# B&R Automation Studio project Tmp_Recipe_V1
Automation Studio 4.9.5.36 SP; technology packages: mapp 5.15.0, mappView 5.15.1

## Configuration X20CPU

CPU X20CP1583, AutomationRuntime C4.90, Build 4.1.2, Safety 0.0, Vc V4.52.0

### Task classes (Cpu.sw)
```
Cyclic#8:
  Recipe_01 <- mappRecipe.Recipe_01.prg
  YourTask <- mappRecipe.YourTask.prg
Binaries: udbdef, mvLoader, TCData, arsvcreg, Config, sysconf, ashwd, ashwac, asfw, iomap, Role, User, arconfig, OpcUaMap
Libraries: FileIO, runtime, AsBrStr, standard, AsBrWStr, MpRecipe, MpBase, sys_lib, IecCheck, AsIODiag, AsHttp, AsMem, MpCom, astime, asieccon
```

### Hardware
```
X20CP1583 : X20CP1583 v1.5.0.0
  Connector IF2:
    ActivateDevice = 1
  ConfigurationID = Tmp_Recipe
  UserPartitionSize = 200
  Simulation = 1
  VolatileGlobalPvSize = 300000
  Cyclic8Stack = 20000
  FileDevice1
  FileDeviceName1 = RECIPE_DEVICE
  FileDevicePath1 = F:/
  FileDevice2
  FileDeviceName2 = SIM_DEVICE
  FileDevicePath2 = C:/Temp
  FtpUser1
  FtpUsername1 = br
  FtpUserPassword1 = B9fKGuUbjkGCgEptWUpgQ1eJbLeEvMYqPBCteWUIcCw=
  FtpUserSalt1 = wEo/3/qm
  FTPAccessRight1 = 0
  ActivateSdm = 0
  ActivateOpcUa = 1
  OpcUaInformationModels_PV_Version = 1
```

### Config_0.mprecipecsv - X20CP1583/mappServices/Config_0.mprecipecsv
```
Element gRecipeCsv_01 (Type=mprecipecsv)
```

### Config_1.mprecipexml - X20CP1583/mappServices/Config_1.mprecipexml
```
Element gRecipeXml_01 (Type=mprecipexml)
```

## Logical view

Binary libraries used (declarations not repeated): AsHttp, AsMem, operator, runtime, astime, AsIecCon, FileIO, AsBrStr, AsBrWStr, standard, MpRecipe 5.07.1, MpBase 5.07.0, sys_lib, AsIODiag, MpCom 5.07.1

### Package Logical/Libraries - Global libraries

### Library Logical/Libraries/IecCheck (IEC)
Depends on: sys_lib, AsBrStr

#### IecCheck.fun - Exported functions and function blocks
```iecst
FUNCTION CheckDivSint : SINT (* Check divisor for SINT division *)
	VAR_INPUT
		divisor : SINT;
	END_VAR
END_FUNCTION

FUNCTION CheckDivUsint : USINT (* Check divisor for USINT division *)
	VAR_INPUT
		divisor : USINT;
	END_VAR
END_FUNCTION

FUNCTION CheckDivInt : INT (* Check divisor for INT division *)
	VAR_INPUT
		divisor : INT;
	END_VAR
END_FUNCTION

FUNCTION CheckDivUint : UINT (* Check divisor for UINT division *)
	VAR_INPUT
		divisor : UINT;
	END_VAR
END_FUNCTION

FUNCTION CheckDivDint : DINT (* Check divisor for DINT division *)
	VAR_INPUT
		divisor : DINT;
	END_VAR
END_FUNCTION

FUNCTION CheckDivUdint : UDINT (* Check divisor for UDINT division *)
	VAR_INPUT
		divisor : UDINT;
	END_VAR
END_FUNCTION

FUNCTION CheckDivReal : REAL (* Check divisor for REAL division *)
	VAR_INPUT
		divisor : REAL;
	END_VAR
END_FUNCTION

FUNCTION CheckDivLReal : LREAL (* Check divisor for LREAL division, not available for SG3 and SGC *)
	VAR_INPUT
		divisor : LREAL;
	END_VAR
END_FUNCTION

FUNCTION CheckBounds : DINT (* Check range for array access *)
	VAR_INPUT
		index : DINT;
		lower : DINT;
		upper : DINT;
	END_VAR
END_FUNCTION

FUNCTION CheckRange : DINT (* Check range for enumeration *)
	VAR_INPUT
		value : DINT;
		lower : DINT;
		upper : DINT;
	END_VAR
END_FUNCTION

FUNCTION CheckSignedSubrange : DINT (* Check range for subrange of signed data types *)
	VAR_INPUT
		value : DINT;
		lower : DINT;
		upper : DINT;
	END_VAR
END_FUNCTION

FUNCTION CheckUnsignedSubrange : UDINT (* Check range for subrange of unsigned data types *)
	VAR_INPUT
		value : UDINT;
		lower : UDINT;
		upper : UDINT;
	END_VAR
END_FUNCTION

FUNCTION CheckReadAccess : UDINT (* Check address when reading dynamic variables *)
	VAR_INPUT
		address : UDINT;
	END_VAR
END_FUNCTION

FUNCTION CheckWriteAccess : UDINT (* Check address when writing dynamic variables *)
	VAR_INPUT
		address : UDINT;
	END_VAR
END_FUNCTION

FUNCTION MakeEntry : UDINT (* Makes an entry (log book entry) in the error log book *)
	VAR
		taskname : STRING[30];
		group : USINT;
		status_name : UINT;
		out_text : STRING[80];
	END_VAR
	VAR_INPUT
		number : UINT;
		index : DINT;
		text : STRING[50];
	END_VAR
END_FUNCTION
```

#### IecCheck.st - Implementation file
```iecst
(* Check divisor for SINT division *)
FUNCTION CheckDivSint
	IF divisor=0 THEN
		CheckDivSint:=1;
		MakeEntry(55555,divisor,'CheckDivSint');
	ELSE
		CheckDivSint:=divisor;
	END_IF
END_FUNCTION

(* Check divisor for USINT division *)
FUNCTION CheckDivUsint
	IF divisor=0 THEN
		CheckDivUsint:=1;
		MakeEntry(55555,divisor,'CheckDivUsint');
	ELSE
		CheckDivUsint:=divisor;
	END_IF
END_FUNCTION

(* Check divisor for INT division *)
FUNCTION CheckDivInt
	IF divisor=0 THEN
		CheckDivInt:=1;
		MakeEntry(55555,divisor,'CheckDivInt');
	ELSE
		CheckDivInt:=divisor;
	END_IF
END_FUNCTION

(* Check divisor for UINT division *)
FUNCTION CheckDivUint
	IF divisor=0 THEN
		CheckDivUint:=1;
		MakeEntry(55555,divisor,'CheckDivUint');
	ELSE
		CheckDivUint:=divisor;
	END_IF
END_FUNCTION

(* Check divisor for DINT division *)
FUNCTION CheckDivDint
	IF divisor=0 THEN
		CheckDivDint:=1;
		MakeEntry(55555,divisor,'CheckDivDint');
	ELSE
		CheckDivDint:=divisor;
	END_IF
END_FUNCTION

(* Check divisor for UDINT division *)
FUNCTION CheckDivUdint
	IF divisor=0 THEN
		CheckDivUdint:=1;
		MakeEntry(55555,divisor,'CheckDivUdint');
	ELSE
		CheckDivUdint:=divisor;
	END_IF
END_FUNCTION

(* Check divisor for REAL division *)
FUNCTION CheckDivReal
	IF divisor=0 THEN
		CheckDivReal:=1;
		MakeEntry(55555,0,'CheckDivReal');
	ELSE
		CheckDivReal:=divisor;
	END_IF
END_FUNCTION

(* Check divisor for LREAL division *)
FUNCTION CheckDivLReal
	IF divisor=0 THEN
		CheckDivLReal:=1;
		MakeEntry(55555,0,'CheckDivLReal');
	ELSE
		CheckDivLReal:=divisor;
	END_IF
END_FUNCTION

(* Check range for array access *)
FUNCTION CheckBounds
	IF index < lower THEN
		CheckBounds := lower;
		MakeEntry(55555,index,'CheckBounds');
	ELSIF index > upper THEN
		CheckBounds := upper;
		MakeEntry(55555,index,'CheckBounds');
	ELSE
		CheckBounds := index;
	END_IF
END_FUNCTION

(* Check range for enumeration *)
FUNCTION CheckRange
	IF value < lower THEN
		CheckRange := lower;
		MakeEntry(55555,value,'CheckRange');
	ELSIF value > upper THEN
		CheckRange := upper;
		MakeEntry(55555,value,'CheckRange');
	ELSE
		CheckRange := value;
	END_IF
END_FUNCTION

(* Check range for subrange of signed data types *)
FUNCTION CheckSignedSubrange
	IF value < lower THEN
		CheckSignedSubrange := lower;
		MakeEntry(55555,value,'CheckSignedSubrange');
	ELSIF value > upper THEN
		CheckSignedSubrange := upper;
		MakeEntry(55555,value,'CheckSignedSubrange');
	ELSE
		CheckSignedSubrange := value;
	END_IF
END_FUNCTION

(* Check range for subrange of unsigned data types *)
FUNCTION CheckUnsignedSubrange
	IF value < lower THEN
		CheckUnsignedSubrange := lower;
		MakeEntry(55555,value,'CheckUnsignedSubrange');
	ELSIF value > upper THEN
		CheckUnsignedSubrange := upper;
		MakeEntry(55555,value,'CheckUnsignedSubrange');
	ELSE
		CheckUnsignedSubrange := value;
	END_IF
END_FUNCTION

(* Check address when reading dynamic variables *)
FUNCTION CheckReadAccess
	IF address=0 THEN
		(* TODO: Insert an appropriate code, see AutomationStudio help for further information *)
		MakeEntry(55555,address,'Read from NULL');
	END_IF

	CheckReadAccess:=0;
END_FUNCTION

(* Check address when writing dynamic variables *)
FUNCTION CheckWriteAccess
	IF address=0 THEN
		(* TODO: Insert an appropriate code, see AutomationStudio help for further information *)
		MakeEntry(55555,address,'Write to NULL');
	END_IF

	CheckWriteAccess:=0;
END_FUNCTION

(* Makes an entry (log book entry) in the error log book *)
FUNCTION MakeEntry
		status_name := ST_name(0,ADR(taskname),ADR(group));

		brsstrcpy(ADR(out_text),ADR(text));
		brsstrcat(ADR(out_text),ADR(' > in task > '));
  		brsstrcat(ADR(out_text),ADR(taskname));
		MakeEntry := ADR(out_text);
		ERRxfatal(number,index,ADR(out_text));
END_FUNCTION
```

- Visualisation Logical/mappView (not shown)

### RecTypes.typ
```iecst
(*------------------------------------------------------------------------------------------------------------------------------------------------------------------------------------------------------------------------*)
(*Global enumerations*)

TYPE
	recSTATE :
		( (*Recipe management state machine*)
		REC_WAIT,
		REC_REG_NAME,
		REC_REG_VAR,
		REC_CREATE_DIR,
		REC_READ_DIR,
		REC_READ_DIR_1,
		REC_READ_DIR_2,
		REC_READ_DIR_3,
		REC_GEN_FILE_NAME,
		REC_LOAD_SAVE,
		REC_DELETE,
		REC_RENAME,
		REC_VIEW,
		REC_DOWNLOAD,
		REC_DOWNLOAD_1,
		REC_DOWNLOAD_2,
		REC_DOWNLOAD_3,
		REC_DOWNLOAD_4,
		REC_UPLOAD,
		REC_UPLOAD_1,
		REC_UPLOAD_2,
		REC_UPLOAD_3,
		REC_UPLOAD_4,
		REC_UPLOAD_5,
		REC_UPLOAD_6,
		REC_ERROR
		);
	recTYPE :
		(
		typeCSV,
		typeXML
		);
END_TYPE

(*------------------------------------------------------------------------------------------------------------------------------------------------------------------------------------------------------------------------*)
(*Global structure*)

TYPE
	recERR : 	STRUCT  (*Recipe management error structure*)
		Text : WSTRING[200]; (* Error text *)
		No : DINT; (* Error number *)
		State : recSTATE; (* Error step *)
	END_STRUCT;
	recCMD : 	STRUCT  (*Recipe management command structure*)
		Init : BOOL := TRUE; (*Init recipes managment*)
		New : BOOL; (*Create new recipe*)
		Load : BOOL; (*Load recipe*)
		Save : BOOL; (*Save recipe*)
		View : BOOL; (*View recipe*)
		Rename : BOOL; (*Rename recipe*)
		Delete : BOOL; (*Delete recipe*)
		Download : BOOL; (*Download recipe*)
		Upload : BOOL; (*Upload recipe*)
		ErrorReset : BOOL; (*Reset pending errors*)
	END_STRUCT;
	recPAR : 	STRUCT  (*Recipe management parameter structure*)
		RecipeName : WSTRING[REC_NAME_LENGTH]; (*Recipe name*)
		RecipeNameNew : WSTRING[REC_NAME_LENGTH]; (*New recipe name*)
		RecipeID : STRING[REC_NAME_LENGTH]; (*File name of the recipe*)
		Initialized : BOOL; (*Indicates that recipe management was initialized*)
		VisuSlotID : USINT; (*ID for connected web connection*)
		VisuEnableCommand : BOOL;
	END_STRUCT;
	recDAT : 	STRUCT  (*Recipe management data structure*)
		RecipeNames : ARRAY[0..REC_REC_NUM]OF WSTRING[REC_NAME_LENGTH]; (*Recipe unicode names*)
		RecipeIDs : ARRAY[0..REC_REC_NUM]OF STRING[REC_NAME_LENGTH]; (*File name of the recipes*)
		RecipeNum : UINT; (*Number of recipes*)
		Status : WSTRING[100]; (*Shows the result of the last command*)
	END_STRUCT;
	recVIS : 	STRUCT  (*Recipe management visualization structure*)
		RecipeNames : ARRAY[0..REC_REC_NUM]OF WSTRING[REC_VIS_LENGTH]; (*Recipe names as mappView data provider*)
		RecipeNum : UINT; (*Number of visible recipes*)
		RecipeFilter : WSTRING[REC_NAME_LENGTH]; (*Only show recipes that fit this pattern*)
		RecipeSelect : WSTRING[REC_NAME_LENGTH]; (*Select recipe in listbox after command new or rename*)
		DownloadFileUrl : STRING[REC_NAME_LENGTH]; (*URL used with recipe download*)
		UploadOverwriteRequest : BOOL; (*Show message box to overwrite file*)
		UploadOverwriteResponse : USINT; (*Response from message box overwrite file*)
		ReloadUpload : BOOL; (*Reload upload button*)
		RecipeDoubleClick : USINT; (*Track double click event*)
		ViewFilePath : STRING[REC_VIS_LENGTH]; (*Full path for viewing file*)
		ViewFile : BOOL; (*Trigger that opens the fly out window when viewing recipes*)
		ShowMessageBoxError : BOOL; (*Show message box on error*)
	END_STRUCT;
	recMAIN : 	STRUCT  (*Recipe management main structure*)
		CMD : recCMD; (* Command structure *)
		PAR : recPAR; (* Parameter structure *)
		DAT : recDAT; (*Data structure*)
		VIS : ARRAY[0..REC_MAX_CLIENTS_ID]OF recVIS; (*Visualization structure*)
		ERR : recERR; (* Error structure *)
	END_STRUCT;
END_TYPE
```

### RecVariables.var
```iecst
(*------------------------------------------------------------------------------------------------------------------------------------------------------------------------------------------------------------------------*)
(*Configuration for recipe managment*)
VAR CONSTANT
	REC_USE_UNICODE : BOOL := FALSE; (*Use standard strings for recipe name when false, use unicode strings for recipe name when true*)
	REC_SORT_NUMERIC : BOOL := FALSE; (*Sort recipe names as numeric values instead of alphabetic*)
	REC_RECIPE_TYPE : recTYPE := typeCSV; (*Type of recipe (CSV / XML)*)
END_VAR
VAR
	REC_MPLINK : {REDUND_UNREPLICABLE} STRING[80] := 'gRecipeCsv_01'; (*mappRecipe link name from configuration view. User gRecipeCsv_01 for CSV and gRecipeXml_01 for XML in this demo*)
END_VAR
VAR CONSTANT
	REC_DEVICE : STRING[80] := 'RECIPE_DEVICE'; (*Device name for the recipe data defined under File Devices in the CPU configuration*)
	REC_DIRECTORY : STRING[80] := 'Recipe_01'; (*Directory where the recipes are stored*)
	REC_THIS_TASK : STRING[40] := 'Recipe_01'; (*Name of this task and the global variables structure*)
	REC_REC_NUM : USINT := 100; (*Maximum number of recipes*)
	REC_VAR_NUM : USINT := 10; (*Maximum number of variables that can be registered*)
	REC_NAME_LENGTH : USINT := 40; (*Maximum length for a recipe name*)
	REC_UPLOAD_DOWNLOAD_SIZE : UDINT := 100000; (*Maximum size of memory allocated for uploading and downloading files*)
	REC_VIS_LENGTH : USINT := 120; (*Make this REC_NAME_LENGTH  x3*)
	REC_MAX_CLIENTS_ID : USINT := 2; (*Highest client ID for concurrent web client connections. Do not change this number.*)
END_VAR
VAR
	REC_VIEW_FILTER : ARRAY[0..9] OF STRING[5] := ['csv','xml',8('')]; (*Files extensions than can be used with the view command*)
END_VAR
(*------------------------------------------------------------------------------------------------------------------------------------------------------------------------------------------------------------------------*)
(*Add you variables to this list*)
VAR
	REC_VAR_LIST : ARRAY[1..REC_VAR_NUM] OF STRING[100] := ['YourTask:MaschineData','YourTask:ProductID','YourTask:CustomerID',7('')]; (*List of variables to be inlcuded in a recipe*)
	Recipe_01 : recMAIN; (*Global recipe structure. The name must match the task name of the recipe managment.*)
END_VAR
```

### Program Logical/mappRecipe/Recipe_01 (IEC)

#### Init.st - Init and local configuration
```iecst
// --------------------------------------------------------------------------------------------------------------------
//	Function:	Recipe management with mappRecipe
//  Version:	0.7
//	Changed:	08.05.2020
// --------------------------------------------------------------------------------------------------------------------

PROGRAM _INIT
	// ----------------------------------------------------------------------------------------
	// The following settings can be adjusted
	IF(DiagCpuIsSimulated()) THEN
		DeviceName 	:= 'SIM_DEVICE';						// Device name from the CPU configuration for simulation
	ELSE
		DeviceName 	:= REC_DEVICE;							// Device name from the CPU configuration for X20CPU
	END_IF

	// ----------------------------------------------------------------------------------------
	// Dont change anything below this line
	// ----------------------------------------------------------------------------------------

	// ----------------------------------------------------------------------------------------
	// Get mapp link information
	MpComGetLink_0.Enable := TRUE;
	MpComGetLink_0.ComponentName := ADR(REC_MPLINK);
	MpComGetLink_0();
	IF(MpComGetLink_0.Error) THEN
	END_IF

	// ----------------------------------------------------------------------------------------
	// Make sure global variable structure and task name are correct
	taskStatus := ST_ident(ADR(REC_THIS_TASK), taskGroup, ADR(taskID));
	pvStatus := PV_xgetadr(ADR(REC_THIS_TASK), ADR(pvADR), ADR(pvLEN));
	// Connect global and local structure
	IF(pvStatus = 0) THEN
		RECIPE ACCESS pvADR;
		brsmemset(ADR(RECIPE.ERR), 0 , SIZEOF(RECIPE.ERR));
		RECIPE.PAR.Initialized := FALSE;
	END_IF

	// ----------------------------------------------------------------------------------------
	// Allocate memory for file upload and download
	AsMemPartCreate_0.enable	:= TRUE;
	AsMemPartCreate_0.len		:= REC_UPLOAD_DOWNLOAD_SIZE;
	AsMemPartCreate_0();
	IF AsMemPartCreate_0.status <> 0 THEN
		rec_state := CreateError(ADR(RECIPE), ERR_MEM_ALLOC, "file upload and download memory alloc failed", rec_state);
	ELSE
		AsMemPartAllocClear_0.enable	:= TRUE;
		AsMemPartAllocClear_0.ident		:= AsMemPartCreate_0.ident;
		AsMemPartAllocClear_0.len		:= REC_UPLOAD_DOWNLOAD_SIZE;
		AsMemPartAllocClear_0();
		IF AsMemPartCreate_0.status <> 0 THEN
			rec_state := CreateError(ADR(RECIPE), ERR_MEM_ALLOC, "file upload and download memory clear failed", rec_state);
		END_IF
	END_IF

	// ----------------------------------------------------------------------------------------
	// Generate HTML messages for web upload
	upload_response	:= '<html><body><form action="/uploadA.html" name="form_upload" method="post" enctype="multipart/form-data" >
	<label for="file-upload" style="font-weight:bold;font-family: sans-serif;font-size:16px;padding:15px 50px;10px;10px;" class="custom-file-upload">Upload</label>
	<input type="file" id="file-upload" style="display:none;" onchange="form.submit()" name="file_selected" content-type="application/octet-stream" />
	</form><body></html> ';
	WebServiceUpload.pServiceName := ADR('uploadA.html');
END_PROGRAM
```

#### Main.st - Cyclic code
```iecst
// --------------------------------------------------------------------------------------------------------------------********
//	Cylic task for recipe management
//	Version 0.7
//	Changed 08.05.2020
// --------------------------------------------------------------------------------------------------------------------********

// --------------------------------------------------------------------------------------------------------------------********
// Cyclic task
// --------------------------------------------------------------------------------------------------------------------********
PROGRAM _CYCLIC
	// --------------------------------------------------------------------------------------------------------------------
	// Make sure task name and global structure correct
	IF(pvStatus <> 0) THEN
		RETURN;
	END_IF
	IF(taskStatus <> 0) THEN
		rec_state := CreateError(ADR(RECIPE), ERR_REC_TASK_NAME, "Task name is incorrect", rec_state);
		RETURN;
	END_IF

	// --------------------------------------------------------------------------------------------------------------------
	// Make sure we dont exceed maximum number of web clients
	IF(RECIPE.PAR.VisuSlotID > REC_MAX_CLIENTS_ID) THEN
		rec_state := CreateError(ADR(RECIPE), ERR_REC_TOO_MANY_CLIENTS, "More than 3 clients try to connect to recipe managment", rec_state);
		RETURN;
	END_IF

	// --------------------------------------------------------------------------------------------------------------------
	// Cyclic function calls
	MpRecipeCsv_0();
	MpRecipeXml_0();

	// ----------------------------------------------------------------------------------------
	// Web service driver for file upload
	WebServiceUpload.enable 			:= TRUE;
	WebServiceUpload.option 			:= httpOPTION_HTTP_11 + httpOPTION_SERVICE_TYPE_NAME;
	WebServiceUpload.pRequestData  		:= AsMemPartAllocClear_0.mem;
	WebServiceUpload.requestDataSize 	:= REC_UPLOAD_DOWNLOAD_SIZE;
	WebServiceUpload.pResponseData 		:= ADR(upload_response);
	WebServiceUpload.responseDataLen 	:= brsstrlen(ADR(upload_response));
	WebServiceUpload();

	// Reset send command
	IF(WebServiceUpload.send = TRUE)  THEN
		WebServiceUpload.send := FALSE;
	// Send response when page is loaded or data is posted
	ELSIF(WebServiceUpload.status = ERR_OK AND WebServiceUpload.send = FALSE) THEN
		WebServiceUpload.send := TRUE;
	// New upload data arrived
	ELSIF(WebServiceUpload.send = FALSE AND WebServiceUpload.requestDataLen > 0 AND RECIPE.CMD.Upload = FALSE) THEN
		// Add delay so that upload can finish
		upload_delay.PT := WebServiceUpload.requestDataLen/100000*5;
		upload_delay.IN := TRUE;
		upload_delay();
	END_IF
	// Check new uploaded data
	IF(upload_delay.Q AND RECIPE.CMD.Upload = FALSE) THEN
		upload_delay.IN := FALSE;
		upload_delay();
		RECIPE.CMD.Upload := TRUE;
	END_IF

	// --------------------------------------------------------------------------------------------------------------------****
	// Recipe management state machine
	// --------------------------------------------------------------------------------------------------------------------****
	CASE rec_state OF
		// --------------------------------------------------------------------------------------------------------------------
		// Wait for command
		// --------------------------------------------------------------------------------------------------------------------
		REC_WAIT:
			// --------------------------------------------------------------------------------------------------------------------
			// Track filter change and data refresh
			IF ((brwcscmp(ADR(RecipeFilterOld[VisuSlotID]), ADR(RECIPE.VIS[VisuSlotID].RecipeFilter)) <> 0) OR (RecipeNumOld[VisuSlotID] <> RECIPE.DAT.RecipeNum)) THEN
				brsmemset(ADR(RECIPE.VIS[VisuSlotID].RecipeNames), 0, SIZEOF(RECIPE.VIS[VisuSlotID].RecipeNames));
				idy := 0;
				IF(RECIPE.DAT.RecipeNum > 0) THEN
					FOR idx:=0 TO RECIPE.DAT.RecipeNum - 1 DO
						// --------------------------------------------------------------------------------
						// Verify that file name contains filter
						IF (brwcslen(ADR(RECIPE.VIS[VisuSlotID].RecipeFilter)) = 0 OR IsInstrW(ADR(RECIPE.DAT.RecipeNames[idx]), ADR(RECIPE.VIS[VisuSlotID].RecipeFilter))) THEN
							WString2DataProvider(ADR(RECIPE.DAT.RecipeNames[idx]), ADR(tmpWStr1));
							RECIPE.VIS[VisuSlotID].RecipeNames[idy] := tmpWStr1;
							idy := idy + 1;
						END_IF
					END_FOR;
					brwcscpy(ADR(RecipeFilterOld[VisuSlotID]), ADR(RECIPE.VIS[VisuSlotID].RecipeFilter));
				END_IF
				RecipeNumOld[VisuSlotID] := RECIPE.DAT.RecipeNum;
				RECIPE.VIS[VisuSlotID].RecipeNum := idy;
			END_IF

			// ------------------------------------------------------------------------------------------------
			// Handle double click for file open
			IF(RECIPE.VIS[VisuSlotID].RecipeDoubleClick > 0) THEN
				DoubleClickRecipeName[VisuSlotID].PT := 50;
				DoubleClickRecipeName[VisuSlotID].IN := TRUE;
				DoubleClickRecipeName[VisuSlotID]();
				// Open selected file
				IF(RECIPE.VIS[VisuSlotID].RecipeDoubleClick > 1) THEN
					DoubleClickRecipeName[VisuSlotID].IN := FALSE;
					DoubleClickRecipeName[VisuSlotID]();
					RECIPE.VIS[VisuSlotID].RecipeDoubleClick := 0;
					RECIPE.PAR.VisuSlotID := VisuSlotID;
					RECIPE.PAR.RecipeName := RECIPE.VIS[VisuSlotID].RecipeSelect;
					RECIPE.CMD.View := TRUE;
				END_IF
			END_IF
			IF(DoubleClickRecipeName[VisuSlotID].Q) THEN
				DoubleClickRecipeName[VisuSlotID].IN := FALSE;
				DoubleClickRecipeName[VisuSlotID]();
				IF(RECIPE.VIS[VisuSlotID].RecipeDoubleClick > 0) THEN
					RECIPE.VIS[VisuSlotID].RecipeDoubleClick := RECIPE.VIS[VisuSlotID].RecipeDoubleClick - 1;
				END_IF
			END_IF

			// Cylce through the client web seesions
			VisuSlotID := VisuSlotID + 1;
			IF(VisuSlotID > REC_MAX_CLIENTS_ID) THEN
				VisuSlotID := 0;
			END_IF

			// --------------------------------------------------------------------------------------------------------------------
			// Disable buttons in visualization when number of recipes is 0
			IF(RECIPE.DAT.RecipeNum = 0) THEN
				RECIPE.PAR.VisuEnableCommand := FALSE;
			ELSE
				RECIPE.PAR.VisuEnableCommand := TRUE;
			END_IF

			// ----------------------------------------------------------------------------------------
			// Reset error reset
			MpRecipeCsv_0.ErrorReset := FALSE;
			MpRecipeXml_0.ErrorReset := FALSE;
			MpRecipeRegPar_0.ErrorReset := FALSE;

			// ----------------------------------------------------------------------------------------
			// Command init/refresh
			IF (RECIPE.CMD.Init = TRUE) THEN
				// Reset data structure and trigger name refresh for vis
				brsmemset(ADR(RECIPE.DAT), 0, SIZEOF(RECIPE.DAT));
				brsmemset(ADR(RecipeIDs), 0, SIZEOF(RecipeIDs));
				brsmemset(ADR(RecipeNumOld), 16#FF, SIZEOF(RecipeNumOld));
				// Skip variable binding if already initialized
				IF(MpRecipeRegPar_1[1].PVName <> 0) THEN
					rec_state := REC_READ_DIR;
				ELSE
					// Register recipe name variable first if unicode is used
					IF(REC_USE_UNICODE) THEN
						rec_state := REC_REG_NAME;
					ELSE
						rec_state := REC_REG_VAR;
					END_IF
					pvCnt := 1;
				END_IF
			// ----------------------------------------------------------------------------------------
			// Command new recipe
			ELSIF (RECIPE.CMD.New = TRUE AND RECIPE.PAR.RecipeName <> "") THEN
				// Show current state
				animation := WorkingStatus(ADR(RECIPE), ADR("creating recipe..."), animation);
				// Verify that we still have space in list
				IF (RECIPE.DAT.RecipeNum > REC_REC_NUM) THEN
					rec_state := CreateError(ADR(RECIPE), ERR_REC_REC_NUM, "maximum number of recipes reached", rec_state);
					RETURN;
				END_IF
				// Make sure recipe does not already exist
				IF(FindRecName(ADR(RECIPE), RECIPE.PAR.RecipeName) <> REC_DOES_NOT_EXIST) THEN
					tmpWStr1 := "recipe name ";
					brwcscat(ADR(tmpWStr1), ADR(RECIPE.PAR.RecipeName));
					brwcscat(ADR(tmpWStr1), ADR(" already exists"));
					rec_state := CreateError(ADR(RECIPE), ERR_REC_NAME_EXISTS, tmpWStr1, rec_state);
					RETURN;
				END_IF
				// Reset selected recipe, copy recipe name to local variable
				RECIPE.VIS[RECIPE.PAR.VisuSlotID].RecipeSelect := "";
				rec_state := REC_GEN_FILE_NAME;
			// ----------------------------------------------------------------------------------------
			// Command load recipe
			ELSIF (RECIPE.CMD.Load = TRUE AND RECIPE.PAR.RecipeName <> "") THEN
				// Show current state
				animation := WorkingStatus(ADR(RECIPE), ADR("loading recipe..."), animation);
				// Copy recipe name to local variable
				rec_state := REC_GEN_FILE_NAME;
				// ----------------------------------------------------------------------------------------
			// Command save recipe
			ELSIF (RECIPE.CMD.Save = TRUE AND (RECIPE.PAR.RecipeName <> "" OR RECIPE.PAR.RecipeNameNew <> "")) THEN
				// Show current state
				animation := WorkingStatus(ADR(RECIPE), ADR("saving recipe..."), animation);
				IF(RECIPE.PAR.RecipeName = "") THEN
					RECIPE.PAR.RecipeName := RECIPE.PAR.RecipeNameNew;
				END_IF
				// Copy recipe name to local variable
				rec_state := REC_GEN_FILE_NAME;
			// ----------------------------------------------------------------------------------------
			// Command view recipe
			ELSIF (RECIPE.CMD.View = TRUE AND RECIPE.PAR.RecipeName <> "") THEN
				// Copy recipe name to local variable
				rec_state := REC_GEN_FILE_NAME;
			// ----------------------------------------------------------------------------------------
			// Command delete recipe
			ELSIF (RECIPE.CMD.Delete = TRUE AND RECIPE.PAR.RecipeName <> "") THEN
				// Show current state, copy recipe name to local variable
				animation := WorkingStatus(ADR(RECIPE), ADR("deleting recipe..."), animation);
				rec_state := REC_GEN_FILE_NAME;
			// ----------------------------------------------------------------------------------------
			// Command download recipe
			ELSIF (RECIPE.CMD.Download = TRUE AND RECIPE.PAR.RecipeName <> "") THEN
				// Show current state, copy recipe name to local variable
				animation := WorkingStatus(ADR(RECIPE), ADR("downloading recipe..."), animation);
				RECIPE.VIS[RECIPE.PAR.VisuSlotID].DownloadFileUrl := '';
				rec_state := REC_GEN_FILE_NAME;
			// ----------------------------------------------------------------------------------------
			// Command upload recipe
			ELSIF (RECIPE.CMD.Upload = TRUE) THEN
				// Make sure that unicode support is turned off
				IF(REC_USE_UNICODE = FALSE) THEN
					// Show current state, copy recipe name to local variable
					animation := WorkingStatus(ADR(RECIPE), ADR("uploading recipe..."), animation);
					rec_state := REC_UPLOAD;
				ELSE
					rec_state := CreateError(ADR(RECIPE), ERR_UNICODE_UPLOAD, "upload is not supported when using unicode recipes", rec_state);
				END_IF
			// ----------------------------------------------------------------------------------------
			// Rename recipe
			ELSIF (RECIPE.CMD.Rename = TRUE AND RECIPE.PAR.RecipeName <> "" AND RECIPE.PAR.RecipeNameNew <> "") THEN
				// Show current state
				animation := WorkingStatus(ADR(RECIPE), ADR("renaming recipe..."), animation);
				// Make sure new recipe name does not already exist
				IF(FindRecName(ADR(RECIPE), RECIPE.PAR.RecipeNameNew) <> REC_DOES_NOT_EXIST) THEN
					tmpWStr1 := "new recipe name ";
					brwcscat(ADR(tmpWStr1), ADR(RECIPE.PAR.RecipeNameNew));
					brwcscat(ADR(tmpWStr1), ADR(" already exists"));
					rec_state := CreateError(ADR(RECIPE), ERR_REC_NAME_EXISTS, tmpWStr1, rec_state);
					RETURN;
				END_IF
				// Reset selected recipe, copy recipe name to local variable
				brsmemset(ADR(RecipeNumOld), 16#FF, SIZEOF(RecipeNumOld));
				RECIPE.VIS[RECIPE.PAR.VisuSlotID].RecipeSelect := "";
				RecipeNameNew := RECIPE.PAR.RecipeNameNew;
				rec_state := REC_GEN_FILE_NAME;
			END_IF
			RecipeName := RECIPE.PAR.RecipeName;

			// ----------------------------------------------------------------------------------------
			// Check parameters
			IF (RECIPE.CMD.Init OR RECIPE.CMD.New OR RECIPE.CMD.Load OR RECIPE.CMD.Save OR RECIPE.CMD.Rename OR RECIPE.CMD.Delete OR RECIPE.CMD.View) THEN
				// Make sure recipe mangament was intialized
				IF (NOT RECIPE.CMD.Init AND NOT RECIPE.PAR.Initialized) THEN
					rec_state := CreateError(ADR(RECIPE), ERR_REC_NOT_INITIALIZED, "recipe management is not initiialized", rec_state);
				END_IF
				// Make sure recipe name is valid
				IF((RECIPE.CMD.New OR RECIPE.CMD.Load OR RECIPE.CMD.Save OR RECIPE.CMD.Rename OR RECIPE.CMD.Delete OR RECIPE.CMD.View) AND RecipeName = "") THEN
					rec_state := CreateError(ADR(RECIPE), ERR_REC_NAME_EMPTY, "recipe name is empty", rec_state);
				END_IF
				// Make sure new recipe name is valid
				IF((RECIPE.CMD.Rename) AND RecipeNameNew = "") THEN
					rec_state := CreateError(ADR(RECIPE), ERR_REC_NAME_EMPTY, "new recipe name is empty", rec_state);
				END_IF
				// Make sure device name is valid
				IF(DeviceName = '') THEN
					rec_state := CreateError(ADR(RECIPE), ERR_REC_DEV_NAME_EMPTY, "device name is empty", rec_state);
				END_IF
				// Make sure variable name has at least one entry
				IF(REC_VAR_LIST[1] = '') THEN
					rec_state := CreateError(ADR(RECIPE), ERR_REC_VAR_NAME_EMPTY, "variable name is empty", rec_state);
				END_IF

				RECIPE.PAR.VisuEnableCommand := FALSE;
			END_IF
		// --------------------------------------------------------------------------------------------------------------------
		// Register recipe name
		// --------------------------------------------------------------------------------------------------------------------
		REC_REG_NAME:
			// Generate string for local recipe name
			tmpStr1 := REC_THIS_TASK;
			brsstrcat(ADR(tmpStr1), ADR(':RecipeName'));

			MpRecipeRegPar_0.Enable := TRUE;
			MpRecipeRegPar_0.MpLink := ADR(MpComGetLink_0.MpLink);
			MpRecipeRegPar_0.PVName := ADR(tmpStr1);
			MpRecipeRegPar_0.Category := ADR(REC_THIS_TASK);

			// ----------------------------------------------------------------------------------------
			// OK
			IF (NOT MpRecipeRegPar_0.Active AND NOT MpRecipeRegPar_0.Error) THEN
				rec_state := REC_REG_VAR;
			// Error
			ELSIF (MpRecipeRegPar_0.Error) THEN
				rec_state := CreateError(ADR(RECIPE), MpRecipeRegPar_0.StatusID, "error trying to register recipe name", rec_state);
			END_IF
		// --------------------------------------------------------------------------------------------------------------------
		// Register variable structure
		// --------------------------------------------------------------------------------------------------------------------
		REC_REG_VAR:
			MpRecipeRegPar_1[pvCnt].Enable := TRUE;
			MpRecipeRegPar_1[pvCnt].MpLink := ADR(MpComGetLink_0.MpLink);
			MpRecipeRegPar_1[pvCnt].PVName := ADR(REC_VAR_LIST[pvCnt]);
			MpRecipeRegPar_1[pvCnt].Category := ADR(REC_THIS_TASK);

			// ----------------------------------------------------------------------------------------
			// OK
			IF (MpRecipeRegPar_1[pvCnt].Active AND NOT MpRecipeRegPar_1[pvCnt].Error) THEN
				pvCnt := pvCnt + 1;
				// Register next variable
				IF((pvCnt >= SIZEOF(REC_VAR_LIST)/SIZEOF(REC_VAR_LIST[pvCnt])) OR (REC_VAR_LIST[pvCnt] = '')) THEN
					rec_state := REC_CREATE_DIR;
				END_IF
			// Error
			ELSIF (MpRecipeRegPar_1[pvCnt].Error) THEN
				tmpWStr1 := "error trying to register variable name ";
				brwcsconv(ADR(tmpWStr2), ADR(REC_VAR_LIST[pvCnt]), brwU8toUC);
				brwcscat(ADR(tmpWStr1), ADR(tmpWStr2));
				rec_state := CreateError(ADR(RECIPE), MpRecipeRegPar_1[pvCnt].StatusID, tmpWStr1, rec_state);
			END_IF
		// --------------------------------------------------------------------------------------------------------------------
		// Create recipe directory
		// --------------------------------------------------------------------------------------------------------------------
		REC_CREATE_DIR:
			DCreate.enable 	:= TRUE;
			DCreate.pDevice	:= ADR(DeviceName);
			DCreate.pName := ADR(REC_DIRECTORY);
			DCreate();

			// ----------------------------------------------------------------------------------------
			// OK
			IF (DCreate.status = OK OR DCreate.status = fiERR_DIR_ALREADY_EXIST) THEN
				// Reset command and return to wait state
				rec_state := REC_READ_DIR;
			// Error
			ELSIF (DCreate.status <> ERR_FUB_BUSY) THEN
				// File device is wrong
				IF(DCreate.status = fiERR_DEVICE_MANAGER) THEN
					rec_state := CreateError(ADR(RECIPE), DCreate.status, "error creating recipe directory, check file device name", rec_state);
				ELSE
					rec_state := CreateError(ADR(RECIPE), DCreate.status, "error creating recipe directory", rec_state);
				END_IF
			END_IF
		// --------------------------------------------------------------------------------------------------------------------
		// Read directory information
		// --------------------------------------------------------------------------------------------------------------------
		REC_READ_DIR:
			// Show current state
			animation := WorkingStatus(ADR(RECIPE), ADR("reading recipes..."), animation);
			// ----------------------------------------------------------------------------------------
			// Clear all entrys
			brsmemset(ADR(RECIPE.DAT), 0, SIZEOF(RECIPE.DAT));
			RECIPE.DAT.RecipeNum := 0;
			// ----------------------------------------------------------------------------------------
			// Set values and get device dir
			DInfo.enable 	:= TRUE;
			DInfo.pDevice	:= ADR(DeviceName);
			DInfo();

			// ----------------------------------------------------------------------------------------
			// OK
			IF (DInfo.status = OK) THEN
				rec_state := REC_READ_DIR_1;
			ELSIF (DInfo.status = fiERR_DEVICE_MANAGER) THEN
				tmpWStr1 := "file device ";
				brwcsconv(ADR(tmpWStr2), ADR(DeviceName), brwU8toUC);
				brwcscat(ADR(tmpWStr1), ADR(tmpWStr2));
				brwcscat(ADR(tmpWStr1), ADR(" is unavailable"));
				rec_state := CreateError(ADR(RECIPE), DInfo.status, tmpWStr1, rec_state);
			ELSIF (DInfo.status = fiERR_DIR_NOT_EXIST) THEN
				tmpWStr1 := "file ";
				brwcsconv(ADR(tmpWStr2), ADR(REC_DIRECTORY), brwU8toUC);
				brwcscat(ADR(tmpWStr1), ADR(tmpWStr2));
				brwcscat(ADR(tmpWStr1), ADR(" is unavailable"));
				rec_state := CreateError(ADR(RECIPE), DInfo.status, tmpWStr1, rec_state);
				// Error
			ELSIF (DInfo.status <> ERR_FUB_BUSY) THEN
				rec_state := CreateError(ADR(RECIPE), DInfo.status, "error dir info", rec_state);
			END_IF
		// --------------------------------------------------------------------------------------------------------------------
		// Open directory
		// --------------------------------------------------------------------------------------------------------------------
		REC_READ_DIR_1:
			DOpen.enable 	:= TRUE;
			DOpen.pDevice	:= ADR(DeviceName);
			DOpen.pName 	:= ADR(REC_DIRECTORY);
			DOpen();

			// ----------------------------------------------------------------------------------------
			// OK
			IF (DOpen.status = OK) THEN
				rec_state := REC_READ_DIR_2;
			// Create error message for missing directory
			ELSIF (DInfo.status = fiERR_DIR_NOT_EXIST) THEN
				tmpWStr1 := "directory ";
				brwcsconv(ADR(tmpWStr2), ADR(REC_DIRECTORY), brwU8toUC);
				brwcscat(ADR(tmpWStr1), ADR(tmpWStr2));
				brwcscat(ADR(tmpWStr1), ADR(" is unavailable"));
				rec_state := CreateError(ADR(RECIPE), DInfo.status, tmpWStr1, rec_state);
			// Error
			ELSIF (DOpen.status <> ERR_FUB_BUSY) THEN
				rec_state := CreateError(ADR(RECIPE), DOpen.status, "error dir open", rec_state);
			END_IF;
		// --------------------------------------------------------------------------------------------------------------------
		// Read file directory information
		// --------------------------------------------------------------------------------------------------------------------
		REC_READ_DIR_2:
			DRead.enable 	:= TRUE;
			DRead.ident		:= DOpen.ident;
			DRead.pData 	:= ADR(lDirReadData);
			DRead.data_len 	:= SIZEOF(lDirReadData);
			DRead();

			// ----------------------------------------------------------------------------------------
			// OK
			IF (DRead.status = OK AND lDirReadData.Mode = fiFILE) THEN
				animation := WorkingStatus(ADR(RECIPE), ADR("initializing recipe managment..."), animation);
				// Make sure file name does not exceed maximum string size
				IF (brsstrlen(ADR(lDirReadData.Filename)) < REC_NAME_LENGTH) THEN
					// Copy dir info to string
					brsmemset(ADR(RECIPE.PAR.RecipeID), 0, SIZEOF(RECIPE.PAR.RecipeID));
					brsstrcpy(ADR(RECIPE.PAR.RecipeID), ADR(lDirReadData.Filename));
					// Make sure file extension is CSV or XML
					IF(brsstrlen(ADR(RECIPE.PAR.RecipeID)) > 4 AND ((REC_RECIPE_TYPE = typeCSV AND brsmemcmp(ADR(RECIPE.PAR.RecipeID) + (brsstrlen(ADR(RECIPE.PAR.RecipeID)) - 4), ADR('.csv'), 4) = 0) OR (REC_RECIPE_TYPE = typeXML AND brsmemcmp(ADR(RECIPE.PAR.RecipeID) + (brsstrlen(ADR(RECIPE.PAR.RecipeID)) - 4), ADR('.xml'), 4) = 0))) THEN
						brsmemset(ADR(RECIPE.PAR.RecipeID) + (brsstrlen(ADR(RECIPE.PAR.RecipeID)) - 4), 0, 4);
						// ------------------------------------------------------------------------------------
						// Verify that we still have space in list
						IF (RECIPE.DAT.RecipeNum <= REC_REC_NUM) THEN
							// --------------------------------------------------------------------
							// Read recipe name from recipe data in next rec_state when using unicode
							IF(REC_USE_UNICODE) THEN
								RecipeIDs[brsatoi(ADR(RECIPE.PAR.RecipeID))] := TRUE;
								rec_state := REC_GEN_FILE_NAME;
								// Generate recipe name from file name
							ELSE
								brwcsconv(ADR(RecipeName), ADR(RECIPE.PAR.RecipeID), brwU8toUC);
								// Generate ASCII data, insert recipe into list
								InsertRecName(ADR(RECIPE), RecipeName, RECIPE.PAR.RecipeID);
							END_IF
							// Error
						ELSE
							rec_state := CreateError(ADR(RECIPE), ERR_REC_REC_NUM, "maximum number of recipes reached", rec_state);
						END_IF
					END_IF
				ELSE
					has_oversized_items := TRUE;
				END_IF
			// Last entry reached
			ELSIF (DRead.status = fiERR_NO_MORE_ENTRIES) THEN
				rec_state := REC_READ_DIR_3;
			// Error
			ELSIF (DRead.status <> ERR_FUB_BUSY AND DRead.status <> OK) THEN
				rec_state := CreateError(ADR(RECIPE), DRead.status, "error recipe list read", rec_state);
			END_IF
		// --------------------------------------------------------------------------------------------------------------------
		// Close directory information
		// --------------------------------------------------------------------------------------------------------------------
		REC_READ_DIR_3:
			DClose.enable 	:= TRUE;
			DClose.ident	:= DOpen.ident;
			DClose();

			// ----------------------------------------------------------------------------------------
			// OK
			IF (DClose.status = OK) THEN
				// Reset command and return to wait state
				RECIPE.DAT.Status := "initializing complete";
				RECIPE.CMD.Init	:= FALSE;
				RECIPE.PAR.RecipeID := '';
				RECIPE.PAR.Initialized := TRUE;
				DClose.ident	:= 0;
				// Create error message for oversized items
				IF(has_oversized_items) THEN
					rec_state := CreateError(ADR(RECIPE), ERR_REC_NAME_LENGTH, "one or more recipe names exceeds maximum length", rec_state);
				ELSE
					rec_state := REC_WAIT;
				END_IF
			// Error
			ELSIF (DClose.status <> ERR_FUB_BUSY) THEN
				rec_state := CreateError(ADR(RECIPE), DClose.status, "error dir close", rec_state);
			END_IF
		// --------------------------------------------------------------------------------------------------------------------
		// Generate recipe name	full path and file name
		// --------------------------------------------------------------------------------------------------------------------
		REC_GEN_FILE_NAME:
			// Find recipe entry
			RecipeIndex := FindRecName(ADR(RECIPE), RecipeName);

			// Generate file name when using unicode strings
			IF(REC_USE_UNICODE) THEN
				// Ignore during init process
				IF(NOT RECIPE.CMD.Init) THEN
					// Find empty slot for new recipe
					IF(RECIPE.CMD.New) THEN
						RecipeIndex := 0;
						WHILE (RecipeIDs[RecipeIndex] = TRUE AND RecipeIndex <= REC_REC_NUM) DO
							RecipeIndex := RecipeIndex + 1;
						END_WHILE;
						// Make sure we found empty slot
						IF(RecipeIndex <= REC_REC_NUM AND RecipeIDs[RecipeIndex] = FALSE) THEN
							brsitoa(RecipeIndex, ADR(RECIPE.PAR.RecipeID));
						ELSE
							rec_state := CreateError(ADR(RECIPE), ERR_REC_REC_NUM, "no empty slot found", rec_state);
							RETURN;
						END_IF
						// Find recipe name in list	for all other command
					ELSE
						// Recipe name was found
						IF(RecipeIndex <> REC_DOES_NOT_EXIST) THEN
							RECIPE.PAR.RecipeID := RECIPE.DAT.RecipeIDs[RecipeIndex];
							// Recipe name was lost
						ELSE
							tmpWStr1 := "recipe name was not found ";
							brwcscat(ADR(tmpWStr1), ADR(RecipeName));
							rec_state := CreateError(ADR(RECIPE), ERR_REC_NAME_LOST, tmpWStr1, rec_state);
							RETURN;
						END_IF
					END_IF
				END_IF
			// Use recipe name as file name when using standard strings
			ELSE
				brwcsconv(ADR(RECIPE.PAR.RecipeID), ADR(RecipeName), brwUCtoU8);
			END_IF

			// Generate recipe path and extension
			RecipeFullFileName := REC_DIRECTORY;
			brsstrcat(ADR(RecipeFullFileName), ADR('/'));
			brsstrcat(ADR(RecipeFullFileName), ADR(RECIPE.PAR.RecipeID));

			// Add file extension
			IF(REC_RECIPE_TYPE = typeCSV) THEN
				brsstrcat(ADR(RecipeFullFileName), ADR('.csv'));
			ELSE
				brsstrcat(ADR(RecipeFullFileName), ADR('.xml'));
			END_IF

			// Save recipe under new name
			IF(RECIPE.CMD.Rename) THEN
				RecipeName := RecipeNameNew;
			END_IF

			// Proceed with next rec_state
			IF(RECIPE.CMD.Delete) THEN
				rec_state := REC_DELETE;
			ELSIF(RECIPE.CMD.View) THEN
				rec_state := REC_VIEW;
			ELSIF(RECIPE.CMD.Rename AND NOT REC_USE_UNICODE) THEN
				rec_state := REC_RENAME;
			ELSIF(RECIPE.CMD.Download) THEN
				rec_state := REC_DOWNLOAD;
			ELSE
				rec_state := REC_LOAD_SAVE;
			END_IF
		// --------------------------------------------------------------------------------------------------------------------
		// Load or save recipe data
		// --------------------------------------------------------------------------------------------------------------------
		REC_LOAD_SAVE:

			IF(REC_RECIPE_TYPE = typeCSV) THEN
				MpRecipeCsv_0.Enable := TRUE;
				MpRecipeCsv_0.MpLink := ADR(MpComGetLink_0.MpLink);
				MpRecipeCsv_0.DeviceName := ADR(DeviceName);
				MpRecipeCsv_0.FileName := ADR(RecipeFullFileName);
				MpRecipeCsv_0.Category := ADR(REC_THIS_TASK);
				MpRecipeCsv_0.Save := RECIPE.CMD.Save OR RECIPE.CMD.New OR RECIPE.CMD.Rename;
				MpRecipeCsv_0.Load := RECIPE.CMD.Load OR RECIPE.CMD.Init;

				MpRecipeDone := MpRecipeCsv_0.CommandDone;
				MpRecipeError := MpRecipeCsv_0.Error;
				MpRecipeStatusID := MpRecipeCsv_0.StatusID;
			ELSE
				MpRecipeXml_0.Enable := TRUE;
				MpRecipeXml_0.MpLink := ADR(MpComGetLink_0.MpLink);
				MpRecipeXml_0.DeviceName := ADR(DeviceName);
				MpRecipeXml_0.FileName := ADR(RecipeFullFileName);
				MpRecipeXml_0.Category := ADR(REC_THIS_TASK);
				MpRecipeXml_0.Save := RECIPE.CMD.Save OR RECIPE.CMD.New OR RECIPE.CMD.Rename;
				MpRecipeXml_0.Load := RECIPE.CMD.Load OR RECIPE.CMD.Init;

				MpRecipeDone := MpRecipeXml_0.CommandDone;
				MpRecipeError := MpRecipeXml_0.Error;
				MpRecipeStatusID := MpRecipeXml_0.StatusID;
			END_IF

			// ----------------------------------------------------------------------------------------
			// OK
			IF (MpRecipeDone AND NOT MpRecipeError AND MpRecipeStatusID = 0) THEN
				// Reset command and return to wait state
				MpRecipeCsv_0.Load := FALSE;
				MpRecipeCsv_0.Save := FALSE;
				MpRecipeXml_0.Load := FALSE;
				MpRecipeXml_0.Save := FALSE;

				// Continue renaming recipe
				IF(RECIPE.CMD.Rename) THEN
					IF(REC_USE_UNICODE) THEN
						// Remove name from recipe list	and add it again
						RemoveRecName(ADR(RECIPE), RecipeIndex);
						InsertRecName(ADR(RECIPE), RecipeName, RECIPE.PAR.RecipeID);

						RECIPE.VIS[RECIPE.PAR.VisuSlotID].RecipeSelect := RecipeName;
						tmpWStr1 := "renamed recipe";
						RECIPE.CMD.Rename := 0;
					ELSE
						rec_state := REC_DELETE;
						RETURN;
					END_IF
				END_IF
				// Continue reading recipe names
				IF(RECIPE.CMD.Init) THEN
					InsertRecName(ADR(RECIPE), RecipeName, RECIPE.PAR.RecipeID);
					rec_state := REC_READ_DIR_2;
					RETURN;
				END_IF
				// Finish new recipe
				IF(RECIPE.CMD.New) THEN
					IF(REC_USE_UNICODE) THEN
						RecipeIDs[brsatoi(ADR(RECIPE.PAR.RecipeID))] := TRUE;
					END_IF
					InsertRecName(ADR(RECIPE), RecipeName, RECIPE.PAR.RecipeID);
					RECIPE.VIS[RECIPE.PAR.VisuSlotID].RecipeSelect := RecipeName;
					tmpWStr1 := "created new recipe";
					RECIPE.CMD.New	:= FALSE;
				END_IF
				// Finish load recipe
				IF(RECIPE.CMD.Load) THEN
					tmpWStr1 := "loaded recipe";
					RECIPE.CMD.Load	:= FALSE;
				END_IF
				// Finish save recipe
				IF(RECIPE.CMD.Save) THEN
					tmpWStr1 := "saved recipe";
					RECIPE.CMD.Save	:= FALSE;
				END_IF
				// Complete status string
				CreateMessage(ADR(RECIPE.DAT.Status), ADR(tmpWStr1), ADR(RecipeName), RECIPE.PAR.VisuSlotID);
				rec_state := REC_WAIT;
			// Error
			ELSIF (MpRecipeStatusID = mpRECIPE_ERR_CONFIG_INVALID) THEN
				rec_state := CreateError(ADR(RECIPE), MpRecipeStatusID, "mapp configuration is invalid, check REC_MPLINK constant", rec_state);
			ELSIF (MpRecipeStatusID = mpRECIPE_WRN_LOAD_WITH_WARN) THEN
				rec_state := CreateError(ADR(RECIPE), MpRecipeStatusID, "warning recipe read/write/new, check PLC logbook for details", rec_state);
			ELSIF (MpRecipeStatusID = mpRECIPE_WRN_NO_PV_FOUND) THEN
				tmpWStr1 := "error recipe file contains no data ";
				brwcsconv(ADR(tmpWStr2), ADR(RecipeFullFileName), brwU8toUC);
				brwcscat(ADR(tmpWStr1), ADR(tmpWStr2));
				rec_state := CreateError(ADR(RECIPE), MpRecipeStatusID, tmpWStr1, rec_state);
			ELSIF (MpRecipeError OR MpRecipeStatusID <> 0) THEN
				tmpWStr1 := "error recipe read/write/new ";
				brwcscat(ADR(tmpWStr1), ADR(RecipeName));
				rec_state := CreateError(ADR(RECIPE), MpRecipeStatusID, tmpWStr1, rec_state);
			END_IF
		// --------------------------------------------------------------------------------------------------------------------
		// Delete selected recipe
		// --------------------------------------------------------------------------------------------------------------------
		REC_DELETE:
			// ----------------------------------------------------------------------------------------
			// Initialize file delete structure
			FDelete.enable		:= TRUE;
			FDelete.pDevice 	:= ADR(DeviceName);
			FDelete.pName		:= ADR(RecipeFullFileName);
			FDelete();

			// ----------------------------------------------------------------------------------------
			// OK
			IF (FDelete.status = OK) THEN
				// Remove name from recipe list
				RemoveRecName(ADR(RECIPE), RecipeIndex);
				// Mark recipe ID as free
				IF(REC_USE_UNICODE) THEN
					RecipeIDs[brsatoi(ADR(RECIPE.PAR.RecipeID))] := FALSE;
				END_IF

				CreateMessage(ADR(RECIPE.DAT.Status), ADR("deleted recipe"), ADR(RecipeName), RECIPE.PAR.VisuSlotID);
				RECIPE.CMD.Delete := 0;
				rec_state := REC_WAIT;
			// Error
			ELSIF (FDelete.status <> ERR_FUB_BUSY) THEN
				tmpWStr1 := "error deleting recipe ";
				brwcscat(ADR(tmpWStr1), ADR(RecipeName));
				rec_state := CreateError(ADR(RECIPE), FDelete.status, tmpWStr1, rec_state);
			END_IF
		// --------------------------------------------------------------------------------------------------------------------
		// Rename selected recipe
		// --------------------------------------------------------------------------------------------------------------------
		REC_RENAME:
			// Generate recipe path and extension
			tmpStr1 := REC_DIRECTORY;
			brsstrcat(ADR(tmpStr1), ADR('/'));
			brwcsconv(ADR(tmpStr2), ADR(RecipeNameNew), brwUCtoU8);
			brsstrcat(ADR(tmpStr1), ADR(tmpStr2));

			// Add file extension
			IF(REC_RECIPE_TYPE = typeCSV) THEN
				brsstrcat(ADR(tmpStr1), ADR('.csv'));
			ELSE
				brsstrcat(ADR(tmpStr1), ADR('.xml'));
			END_IF

			// ----------------------------------------------------------------------------------------
			// Initialize file delete structure
			FRename.enable		:= TRUE;
			FRename.pDevice 	:= ADR(DeviceName);
			FRename.pName		:= ADR(RecipeFullFileName);
			FRename.pNewName	:= ADR(tmpStr1);
			FRename();

			// ----------------------------------------------------------------------------------------
			// OK
			IF (FRename.status = OK) THEN
				// Remove name from recipe list	and add it again
				brsmemmove(ADR(RECIPE.DAT.RecipeNames[RecipeIndex]),ADR(RECIPE.DAT.RecipeNames[RecipeIndex+1]), (RECIPE.DAT.RecipeNum) * SIZEOF(RECIPE.DAT.RecipeNames[0]));
				brsmemmove(ADR(RECIPE.DAT.RecipeIDs[RecipeIndex]),ADR(RECIPE.DAT.RecipeIDs[RecipeIndex+1]), (RECIPE.DAT.RecipeNum) * SIZEOF(RECIPE.DAT.RecipeIDs[0]));
				RECIPE.DAT.RecipeNum := RECIPE.DAT.RecipeNum - 1;

				// Use the same name for unicode
				IF(REC_USE_UNICODE) THEN
					InsertRecName(ADR(RECIPE), RecipeNameNew, RECIPE.PAR.RecipeID);
				// Use the new name for ASCII
				ELSE
					InsertRecName(ADR(RECIPE), RecipeNameNew, tmpStr2);
				END_IF

				RECIPE.VIS[RECIPE.PAR.VisuSlotID].RecipeSelect := RecipeNameNew;
				CreateMessage(ADR(RECIPE.DAT.Status), ADR("renamed recipe"), ADR(RecipeName), RECIPE.PAR.VisuSlotID);
				RECIPE.CMD.Rename := FALSE;
				rec_state := REC_WAIT;
			// Error
			ELSIF (FRename.status <> ERR_FUB_BUSY) THEN
				tmpWStr1 := "error renaming recipe ";
				brwcscat(ADR(tmpWStr1), ADR(RecipeName));
				rec_state := CreateError(ADR(RECIPE), FRename.status, tmpWStr1, rec_state);
			END_IF
		// --------------------------------------------------------------------------------------------------------------------
		// View selected file
		// --------------------------------------------------------------------------------------------------------------------
		REC_VIEW:
			IF(RECIPE.DAT.RecipeNum > 0) THEN
				FOR idx:=0 TO SIZEOF(REC_VIEW_FILTER)/SIZEOF(REC_VIEW_FILTER[0]) - 1 DO
					IF(brsstrlen(ADR(RecipeFullFileName)) >= brsstrlen(ADR(REC_VIEW_FILTER[idx])) AND REC_VIEW_FILTER[idx] <> '') THEN
						// --------------------------------------------------------------------------------
						// Verify that file name contains filter
						IF(brsmemcmp(ADR(RecipeFullFileName) + brsstrlen(ADR(RecipeFullFileName)) - brsstrlen(ADR(REC_VIEW_FILTER[idx])) , ADR(REC_VIEW_FILTER[idx]), brsstrlen(ADR(REC_VIEW_FILTER[idx]))) = 0) THEN
							RECIPE.VIS[RECIPE.PAR.VisuSlotID].ViewFilePath := '/FileDevice:';
							brsstrcat(ADR(RECIPE.VIS[RECIPE.PAR.VisuSlotID].ViewFilePath), ADR(DeviceName));
							brsstrcat(ADR(RECIPE.VIS[RECIPE.PAR.VisuSlotID].ViewFilePath), ADR("/"));
							brsstrcat(ADR(RECIPE.VIS[RECIPE.PAR.VisuSlotID].ViewFilePath), ADR(RecipeFullFileName));
							RECIPE.CMD.View := FALSE;
							RECIPE.VIS[RECIPE.PAR.VisuSlotID].ViewFile := TRUE;
							rec_state := REC_WAIT;
							RETURN;
						END_IF
					END_IF
				END_FOR;
				RECIPE.DAT.Status := "error this file extension is not supported for viewing";
				RECIPE.CMD.View := FALSE;
				rec_state := REC_WAIT;
			END_IF
		// --------------------------------------------------------------------------------------------------------------------
		// Download recipe - open recipe file
		// --------------------------------------------------------------------------------------------------------------------
		REC_DOWNLOAD:
			// ----------------------------------------------------------------------------------------
			// Initialize file open structure
			FOpen.enable	:= TRUE;
			FOpen.pDevice 	:= ADR(DeviceName);
			FOpen.pFile		:= ADR(RecipeFullFileName);
			FOpen();

			// ----------------------------------------------------------------------------------------
			// OK
			IF (FOpen.status = OK) THEN
				// Make sure file fits into memory
				IF(FOpen.filelen <= REC_UPLOAD_DOWNLOAD_SIZE) THEN
					// Clear memory and reset web service
					brsmemset(AsMemPartAllocClear_0.mem, 0, REC_UPLOAD_DOWNLOAD_SIZE);
					WebserviceDownload.enable := FALSE;
					WebserviceDownload();
					rec_state := REC_DOWNLOAD_1;
					// File is too large
				ELSE
					tmpWStr1 := "download file exceeds maximum buffer size of ";
					brsitoa(REC_UPLOAD_DOWNLOAD_SIZE, ADR(tmpStr2));
					brsstrcat(ADR(tmpWStr1), ADR(tmpWStr2));
					brsstrcat(ADR(tmpWStr1), ADR(" bytes"));
					rec_state := CreateError(ADR(RECIPE), ERR_MEM_DOWNLOAD, tmpWStr1, rec_state);
				END_IF;
			// Error
			ELSIF (FOpen.status <> ERR_FUB_BUSY) THEN
				rec_state := CreateError(ADR(RECIPE), FOpen.status, "error opening file for download", rec_state);
			END_IF
		// --------------------------------------------------------------------------------------------------------------------
		// Download recipe - read recipe file
		// --------------------------------------------------------------------------------------------------------------------
		REC_DOWNLOAD_1:
			// ----------------------------------------------------------------------------------------
			// Initialize file read structure
			FRead.enable	:= TRUE;
			FRead.ident		:= FOpen.ident;
			FRead.len		:= FOpen.filelen;
			FRead.pDest		:= AsMemPartAllocClear_0.mem;
			FRead();

			// ----------------------------------------------------------------------------------------
			// OK
			IF (FRead.status = OK) THEN
				rec_state := REC_DOWNLOAD_2;
			// Error
			ELSIF (FRead.status <> ERR_FUB_BUSY) THEN
				rec_state := CreateError(ADR(RECIPE), FRead.status, "error reading file for download", rec_state);
			END_IF
		// --------------------------------------------------------------------------------------------------------------------
		// Download recipe - close recipe file
		// --------------------------------------------------------------------------------------------------------------------
		REC_DOWNLOAD_2:
			// ----------------------------------------------------------------------------------------
			// Initialize file close structure
			FClose.enable	:= TRUE;
			FClose.ident	:= FOpen.ident;
			FClose();

			// ----------------------------------------------------------------------------------------
			// OK
			IF (FClose.status = OK) THEN
				download_timeout.IN := 0;
				download_timeout();
				rec_state := REC_DOWNLOAD_3;
			// Error
			ELSIF (FClose.status <> ERR_FUB_BUSY) THEN
				rec_state := CreateError(ADR(RECIPE), FClose.status, "error closing file for download", rec_state);
			END_IF
		// --------------------------------------------------------------------------------------------------------------------
		// Download recipe - web service
		// --------------------------------------------------------------------------------------------------------------------
		REC_DOWNLOAD_3:
			// ----------------------------------------------------------------------------------------
			// Create response header
			response_header_data :=  'Content-Type: application/octet-stream; Content-Transfer-Encoding: binary; Content-Disposition: attachment; filename="';
			brwcsconv(ADR(tmpStr1), ADR(RecipeName), brwUCtoU8);
			// Add file extension to file name
			IF(REC_RECIPE_TYPE = typeCSV) THEN
				brsstrcat(ADR(tmpStr1), ADR('.csv'));
			ELSE
				brsstrcat(ADR(tmpStr1), ADR('.xml'));
			END_IF
			ReplaceString(ADR(tmpStr1), ADR(' '), ADR('%20'), FALSE);
			brsstrcat(ADR(response_header_data), ADR(tmpStr1));
			brsstrcat(ADR(response_header_data), ADR('"'));

			// ----------------------------------------------------------------------------------------
			// Pre-configure web service for download
			response_header.rawHeader.pData 	:= ADR(response_header_data);
			response_header.rawHeader.dataSize 	:= SIZEOF(response_header_data);
			response_header.rawHeader.dataLen 	:= brsstrlen(ADR(response_header_data));

			// ----------------------------------------------------------------------------------------
			// Start web service
			WebserviceDownload.enable 			:= TRUE;
			WebserviceDownload.option 			:= httpOPTION_HTTP_10 + httpOPTION_SERVICE_TYPE_NAME;
			WebserviceDownload.pResponseData 	:= AsMemPartAllocClear_0.mem;
			WebserviceDownload.pResponseHeader	:= ADR(response_header);
			WebserviceDownload.pServiceName 	:= ADR(tmpStr1);
			WebserviceDownload.responseDataLen 	:= FOpen.filelen;
			WebserviceDownload();

			// ----------------------------------------------------------------------------------------
			// Timeout if file is not pulled from browser
			download_timeout.IN := TRUE;
			download_timeout.PT := 300;
			download_timeout();
			IF(download_timeout.Q) THEN
				rec_state := CreateError(ADR(RECIPE), ERR_TIMEOUT_DOWNLOAD, "error download response timed out", rec_state);
			END_IF

			// ----------------------------------------------------------------------------------------
			// Set URL
			IF (WebserviceDownload.status = ERR_FUB_BUSY AND RECIPE.VIS[RECIPE.PAR.VisuSlotID].DownloadFileUrl = '') THEN
				brsstrcat(ADR(RECIPE.VIS[RECIPE.PAR.VisuSlotID].DownloadFileUrl), ADR(tmpStr1));
			// Start sending data
			ELSIF (WebserviceDownload.status = OK AND WebserviceDownload.send = FALSE AND RECIPE.VIS[RECIPE.PAR.VisuSlotID].DownloadFileUrl <> '') THEN
				WebserviceDownload.send := TRUE;
			// Sending data finished
			ELSIF (WebserviceDownload.send = TRUE) THEN
				WebserviceDownload.send := FALSE;
				rec_state := REC_DOWNLOAD_4;
			// Error
			ELSIF (WebserviceDownload.status <> ERR_FUB_BUSY AND WebserviceDownload.status <> OK) THEN
				rec_state := CreateError(ADR(RECIPE), WebserviceDownload.status, "error sending web response", rec_state);
			END_IF
		// --------------------------------------------------------------------------------------------------------------------
		// Download recipe - web service
		// --------------------------------------------------------------------------------------------------------------------
		REC_DOWNLOAD_4:
			WebserviceDownload();

			// ----------------------------------------------------------------------------------------
			// Start sending data
			IF (WebserviceDownload.phase = httpPHASE_WAITING) THEN
				CreateMessage(ADR(RECIPE.DAT.Status), ADR("downloaded recipe"), ADR(RecipeName), RECIPE.PAR.VisuSlotID);
				RECIPE.VIS[RECIPE.PAR.VisuSlotID].DownloadFileUrl := '';
				WebserviceDownload.send := FALSE;
				RECIPE.CMD.Download := FALSE;
				rec_state := REC_WAIT;
			// Error
			ELSIF (WebserviceDownload.status <> ERR_FUB_BUSY) THEN
				rec_state := CreateError(ADR(RECIPE), WebserviceDownload.status, "error sending web response", rec_state);
			END_IF
		//**********************************************************************************************
		// Upload file - verify parameters
		//**********************************************************************************************
		REC_UPLOAD:

			// Make sure data fits into memory
			IF(WebServiceUpload.requestDataLen < REC_UPLOAD_DOWNLOAD_SIZE) THEN
				// Find file name start
				file_name_start := FindInMem(AsMemPartAllocClear_0.mem, WebServiceUpload.requestDataLen, ADR('filename="'), brsstrlen(ADR('filename="'))) + brsstrlen(ADR('filename="'));
				IF(file_name_start > 0) THEN
					// Find end of file name
					file_name_len := FindInMem(AsMemPartAllocClear_0.mem+file_name_start, WebServiceUpload.requestDataLen-file_name_start, ADR('"$r$n'), brsstrlen(ADR('"$r$n')));
					IF(file_name_len > 0) THEN
						// Make sure file name is not too long
						IF(file_name_len <= SIZEOF(item_name)) THEN
							// Store file name
							brsmemset(ADR(item_name), 0, SIZEOF(item_name));
							brsmemcpy(ADR(item_name), AsMemPartAllocClear_0.mem+file_name_start, file_name_len);
							// Find start of data
							file_data_start := FindInMem(AsMemPartAllocClear_0.mem, WebServiceUpload.requestDataLen, ADR('Content-Type:'), brsstrlen(ADR('Content-Type:'))) + brsstrlen(ADR('Content-Type:'));
							IF(file_data_start > 0) THEN
								// Find end of data
								file_data_start := FindInMem(AsMemPartAllocClear_0.mem+file_data_start, WebServiceUpload.requestDataLen-file_data_start, ADR('$r$n$r$n'), brsstrlen(ADR('$r$n$r$n'))) + brsstrlen(ADR('$r$n$r$n'))+file_data_start;
								file_data_len := FindInMem(AsMemPartAllocClear_0.mem+file_data_start, WebServiceUpload.requestDataLen-file_data_start, ADR('$r$n------'), brsstrlen(ADR('$r$n------')));
								// When file name and data is correct procceed with saving data to file
								IF(file_data_len > 0) THEN
									rec_state := REC_UPLOAD_1;
									RETURN;
								ELSE
									rec_state := CreateError(ADR(RECIPE), ERR_SIZE_DATA_UPLOAD, "data end not found in upload response", rec_state);
								END_IF
							// Data start not found in upload response
							ELSE
								rec_state := CreateError(ADR(RECIPE), ERR_POS_DATA_UPLOAD, "data start not found in upload response", rec_state);
							END_IF
						// File name is too long in upload response
						ELSE
							rec_state := CreateError(ADR(RECIPE), ERR_LEN_NAME_UPLOAD, "file name is too long in upload response", rec_state);
						END_IF
					// File name end not found in upload response
					ELSE
						rec_state := CreateError(ADR(RECIPE), ERR_SIZE_NAME_UPLOAD, "file name end not found in upload response", rec_state);
					END_IF
				// File name start not found in upload response
				ELSE
					rec_state := CreateError(ADR(RECIPE), ERR_POS_NAME_UPLOAD, "file name position not found in upload response", rec_state);
				END_IF
			// Upload file exceeds maximum buffer size
			ELSE
				tmpWStr1 := "upload file exceeds maximum buffer size of ";
				brsitoa(REC_UPLOAD_DOWNLOAD_SIZE, ADR(tmpStr2));
				brsstrcat(ADR(tmpWStr1), ADR(tmpWStr2));
				brsstrcat(ADR(tmpWStr1), ADR(" bytes"));
				rec_state := CreateError(ADR(RECIPE), ERR_MEM_UPLOAD, tmpWStr1, rec_state);
			END_IF
			// Reset upload buffer and function block
			brsmemset(AsMemPartAllocClear_0.mem, 0, REC_UPLOAD_DOWNLOAD_SIZE);
			RECIPE.VIS[RECIPE.PAR.VisuSlotID].ReloadUpload := TRUE;
			WebServiceUpload.enable := FALSE;
			WebServiceUpload();
		//**********************************************************************************************
		// Upload file - Check if file exists
		//**********************************************************************************************
		REC_UPLOAD_1:
			// ----------------------------------------------------------------------------------------
			// Checking for files with the same name
			RECIPE.VIS[RECIPE.PAR.VisuSlotID].UploadOverwriteResponse := 0;
			tmpStr1 := item_name;
			ReplaceString(ADR(tmpStr1), ADR('.csv'), ADR(''), TRUE);
			ReplaceString(ADR(tmpStr1), ADR('.xml'), ADR(''), TRUE);

			FOR idx:=0 TO RECIPE.DAT.RecipeNum DO
				IF(RECIPE.CMD.Upload = TRUE AND RECIPE.DAT.RecipeIDs[idx] = tmpStr1) THEN
					RECIPE.VIS[RECIPE.PAR.VisuSlotID].UploadOverwriteRequest := TRUE;
					rec_state := REC_UPLOAD_2;
					RETURN;
				END_IF;
			END_FOR;

			// Generate recipe path and extension
			RecipeFullFileName := REC_DIRECTORY;
			brsstrcat(ADR(RecipeFullFileName), ADR('/'));
			brsstrcat(ADR(RecipeFullFileName), ADR(item_name));
			rec_state := REC_UPLOAD_4;
		//**********************************************************************************************
		// Upload file - Wait for message box response
		//**********************************************************************************************
		REC_UPLOAD_2:
			// Overwrite file
			IF(RECIPE.VIS[RECIPE.PAR.VisuSlotID].UploadOverwriteResponse = YES) THEN
				RECIPE.VIS[RECIPE.PAR.VisuSlotID].UploadOverwriteRequest := FALSE;
				// Generate recipe path and extension
				RecipeFullFileName := REC_DIRECTORY;
				brsstrcat(ADR(RecipeFullFileName), ADR('/'));
				brsstrcat(ADR(RecipeFullFileName), ADR(item_name));

				rec_state := REC_UPLOAD_3;
			// Do not overwrite file
			ELSIF(RECIPE.VIS[RECIPE.PAR.VisuSlotID].UploadOverwriteResponse = NO) THEN
				// Reset upload command
				brsmemset(AsMemPartAllocClear_0.mem, 0, REC_UPLOAD_DOWNLOAD_SIZE);
				WebServiceUpload.enable := FALSE;
				WebServiceUpload();
				RECIPE.CMD.Upload := 0;
				RECIPE.VIS[RECIPE.PAR.VisuSlotID].ReloadUpload := TRUE;
				RECIPE.VIS[RECIPE.PAR.VisuSlotID].UploadOverwriteRequest	:= FALSE;
				rec_state := REC_WAIT;
			END_IF
		// --------------------------------------------------------------------------------------------------------------------
		// Upload recipe - delete existing recipe
		// --------------------------------------------------------------------------------------------------------------------
		REC_UPLOAD_3:
			// ----------------------------------------------------------------------------------------
			// Initialize file delete structure
			FDelete.enable		:= TRUE;
			FDelete.pDevice 	:= ADR(DeviceName);
			FDelete.pName		:= ADR(RecipeFullFileName);
			FDelete();

			// ----------------------------------------------------------------------------------------
			// OK
			IF (FDelete.status = OK) THEN
				rec_state := REC_UPLOAD_4;
			// Error
			ELSIF (FDelete.status <> ERR_FUB_BUSY) THEN
				tmpWStr1 := "error deleting recipe ";
				brwcscat(ADR(tmpWStr1), ADR(RecipeName));
				rec_state := CreateError(ADR(RECIPE), FDelete.status, tmpWStr1, rec_state);
			END_IF
			//**********************************************************************************************
			// Upload file
			//**********************************************************************************************
		REC_UPLOAD_4:
			// ----------------------------------------------------------------------------------------
			// Initialize file create structure
			FCreate.enable	:= TRUE;
			FCreate.pDevice := ADR(DeviceName);
			FCreate.pFile	:= ADR(RecipeFullFileName);
			FCreate();

			// ----------------------------------------------------------------------------------------
			// OK
			IF (FCreate.status = OK) THEN
				rec_state := REC_UPLOAD_5;
			// Error
			ELSIF (FCreate.status <> ERR_FUB_BUSY) THEN
				rec_state := CreateError(ADR(RECIPE), FCreate.status, "error creating file from upload", rec_state);
				// Reset upload buffer and function block
				brsmemset(AsMemPartAllocClear_0.mem, 0, REC_UPLOAD_DOWNLOAD_SIZE);
				RECIPE.VIS[RECIPE.PAR.VisuSlotID].ReloadUpload := TRUE;
				WebServiceUpload.enable := FALSE;
				WebServiceUpload();
				FCreate.enable	:= FALSE;
				FCreate();
			END_IF
		//**********************************************************************************************
		// Upload file
		//**********************************************************************************************
		REC_UPLOAD_5:

			// ----------------------------------------------------------------------------------------
			// Initialize file write structure
			FWrite.enable	:= TRUE;
			FWrite.ident	:= FCreate.ident;
			FWrite.len		:= file_data_len;
			FWrite.pSrc		:= AsMemPartAllocClear_0.mem + file_data_start;
			FWrite();

			// ----------------------------------------------------------------------------------------
			// OK
			IF (FWrite.status = OK) THEN
				rec_state := REC_UPLOAD_6;
			// Error
			ELSIF (FWrite.status <> ERR_FUB_BUSY) THEN
				rec_state := CreateError(ADR(RECIPE), FWrite.status, "error writing file from upload", rec_state);
			END_IF
		//**********************************************************************************************
		// Upload file
		//**********************************************************************************************
		REC_UPLOAD_6:
			// ----------------------------------------------------------------------------------------
			// Initialize file close structure
			FClose.enable	:= TRUE;
			FClose.ident	:= FCreate.ident;
			FClose();

			// ----------------------------------------------------------------------------------------
			// OK
			IF (FClose.status = OK) THEN
				brsmemset(AsMemPartAllocClear_0.mem, 0, REC_UPLOAD_DOWNLOAD_SIZE);
				WebServiceUpload.enable := FALSE;
				WebServiceUpload();
				RECIPE.CMD.Upload := FALSE;
				RECIPE.CMD.Init := TRUE;
				RECIPE.VIS[RECIPE.PAR.VisuSlotID].ReloadUpload := TRUE;
				rec_state := REC_WAIT;
			// Error
			ELSIF (FClose.status <> ERR_FUB_BUSY) THEN
				rec_state := CreateError(ADR(RECIPE), FClose.status, "error closing file from upload", rec_state);
			END_IF
		// --------------------------------------------------------------------------------------------------------------------
		// Error
		// --------------------------------------------------------------------------------------------------------------------
		REC_ERROR:
			RECIPE.DAT.Status := "error state triggered on web client ID ";
			tmpWStr1 := DINT_TO_WSTRING(RECIPE.PAR.VisuSlotID);
			brwcscat(ADR(RECIPE.DAT.Status), ADR(tmpWStr1));
			// --------------------------------------------------------------------------------------------------------------------
			// Make sure we dont exceed maximum number of web clients
			IF(RECIPE.PAR.VisuSlotID <= REC_MAX_CLIENTS_ID) THEN
				RECIPE.VIS[RECIPE.PAR.VisuSlotID].ShowMessageBoxError := TRUE;
			END_IF
			// --------------------------------------------------------------------------------------------------------------------
			// Return to idle state
			IF RECIPE.CMD.ErrorReset THEN
				// Clear download memory and reset web service
				brsmemset(AsMemPartAllocClear_0.mem, 0, REC_UPLOAD_DOWNLOAD_SIZE);
				WebserviceDownload.enable := FALSE;
				WebserviceDownload();
				WebServiceUpload.enable := FALSE;
				WebServiceUpload();
				RECIPE.VIS[RECIPE.PAR.VisuSlotID].UploadOverwriteRequest := FALSE;

				// Reset function blocks
				MpRecipeCsv_0.ErrorReset := TRUE;
				MpRecipeCsv_0.Save := FALSE;
				MpRecipeCsv_0.Load := FALSE;

				MpRecipeXml_0.ErrorReset := TRUE;
				MpRecipeXml_0.Save := FALSE;
				MpRecipeXml_0.Load := FALSE;

				MpRecipeRegPar_0.ErrorReset := TRUE;

				// Reset error structure
				brsmemset(ADR(RECIPE.ERR), 0, SIZEOF(RECIPE.ERR));
				RECIPE.DAT.Status := "";
				RECIPE.CMD.ErrorReset := FALSE;
				RECIPE.VIS[RECIPE.PAR.VisuSlotID].ShowMessageBoxError := FALSE;
				rec_state := REC_WAIT;
			END_IF;
			brsmemset(ADR(RECIPE.CMD), 0, SIZEOF(RECIPE.CMD));
			RETURN;
	END_CASE
	// --------------------------------------------------------------------------------------------------------------------
	// Cyclic function calls
	MpRecipeRegPar_0();
	FOR idx:=1 TO REC_VAR_NUM DO
		MpRecipeRegPar_1[idx]();
		IF(REC_VAR_LIST[idx] = '') THEN
			EXIT;
		END_IF
	END_FOR;
	MpRecipeCsv_0();
	MpRecipeXml_0();

END_PROGRAM
```

#### Exit.st
```iecst
PROGRAM _EXIT
	// --------------------------------------------------------------------------------------------------------------------
	// Cyclic function calls
	MpRecipeRegPar_0(Enable := FALSE);
	FOR pvCnt:=1 TO REC_VAR_NUM DO
		MpRecipeRegPar_1[pvCnt](Enable := FALSE);
		IF(REC_VAR_LIST[pvCnt] = '') THEN
			EXIT;
		END_IF
	END_FOR;
	MpRecipeCsv_0(Enable := FALSE);
	MpRecipeXml_0(Enable := FALSE);

END_PROGRAM
```

#### RecipeVariables.var - Local variables
```iecst
(*------------------------------------------------------------------------------------------------------------------------------------------------------------------------------------------------------------------------*)
(*Local constants*)
VAR CONSTANT
	OK : USINT := 0; (*Constant for status OK *)
	REC_DOES_NOT_EXIST : UINT := 65535; (*Constant for record does not exist*)
	YES : USINT := 1;
	NO : USINT := 2;
END_VAR
(*------------------------------------------------------------------------------------------------------------------------------------------------------------------------------------------------------------------------*)
(*Local Variables*)
VAR
	RECIPE : REFERENCE TO recMAIN; (*Local recipe structure*)
	DeviceName : STRING[80];
	RecipeIDs : ARRAY[0..REC_REC_NUM] OF BOOL; (*Used with unicode option, keeps tracks of the IDs used*)
	RecipeIndex : UINT; (*Current recipe index*)
	RecipeName : WSTRING[REC_NAME_LENGTH]; (*Local recipe name*)
	RecipeNameNew : WSTRING[REC_NAME_LENGTH]; (*Local recipe new name*)
	RecipeFullFileName : STRING[200]; (*Full recipe name*)
	RecipeFilterOld : ARRAY[0..REC_MAX_CLIENTS_ID] OF WSTRING[REC_NAME_LENGTH]; (*Track filter change *)
	RecipeNumOld : ARRAY[0..REC_MAX_CLIENTS_ID] OF UINT;
	rec_state : recSTATE := REC_WAIT; (*Main step index *)
	animation : USINT := 0; (*Animation for working status	*)
	VisuSlotID : USINT; (*Slot of the visualization that is current used*)
	idx : UINT; (*Index*)
	idy : UINT; (*Index*)
	has_oversized_items : BOOL; (*Indicates that at least one recipe name exceeds the maximum length*)
	tmpStr1 : STRING[200]; (*Temporary string variable *)
	tmpStr2 : STRING[200]; (*Temporary string variable *)
	tmpWStr1 : WSTRING[REC_VIS_LENGTH]; (*Temporary unicode string variable *)
	tmpWStr2 : WSTRING[REC_VIS_LENGTH]; (*Temporary unicode string variable *)
	lDirReadData : fiDIR_READ_EX_DATA; (*File information structure*)
	this : STRING[100]; (*Name of the task and global recipe structure*)
	taskID : UDINT; (*Task ID*)
	taskGroup : USINT; (*Task Group*)
	taskStatus : UINT; (*Status of task information*)
	pvADR : UDINT; (*Adress of global variable structure*)
	pvLEN : UDINT; (*Lenght of global variable structure*)
	pvStatus : UINT; (*Status of global variable information*)
	pvCnt : UINT;
	MpRecipeDone : BOOL; (*Generic status done*)
	MpRecipeError : BOOL; (*Genereic status error*)
	MpRecipeStatusID : DINT; (*Generic error details*)
	DoubleClickRecipeName : ARRAY[0..REC_MAX_CLIENTS_ID] OF TON_10ms; (*Timer for double click detection*)
	response_header : httpResponseHeader_t; (*Response header for download*)
	response_header_data : STRING[300]; (*Response header data*)
	upload_delay : TON_10ms; (*Wait for upload data to finish*)
	download_timeout : TON_10ms; (*Timeout when download must finish*)
	upload_response : STRING[600]; (*Response for upload*)
	file_name_start : UDINT; (*Start of file name in upload data*)
	file_name_len : UDINT; (*Length of file name in upload data*)
	file_data_start : UDINT; (*Start of data in upload data*)
	file_data_len : UDINT; (*Length of data in upload data*)
	item_name : STRING[REC_NAME_LENGTH]; (*Recipe name in upload data*)
END_VAR
(*------------------------------------------------------------------------------------------------------------------------------------------------------------------------------------------------------------------------*)
(*Local function calls*)
VAR
	DInfo : DirInfo;
	DOpen : DirOpen;
	DRead : DirReadEx;
	DClose : DirClose;
	DCreate : DirCreate;
	FOpen : FileOpen;
	FCreate : FileCreate;
	FRead : FileReadEx;
	FWrite : FileWrite;
	FClose : FileClose;
	FDelete : FileDelete;
	FRename : FileRename;
	WebserviceDownload : httpService := (0);
	WebServiceUpload : httpService := (0);
	AsMemPartCreate_0 : AsMemPartCreate;
	AsMemPartAllocClear_0 : AsMemPartAllocClear;
	MpRecipeCsv_0 : MpRecipeCsv;
	MpRecipeXml_0 : MpRecipeXml;
	MpRecipeRegPar_0 : MpRecipeRegPar;
	MpRecipeRegPar_1 : ARRAY[1..REC_VAR_NUM] OF MpRecipeRegPar;
	MpComGetLink_0 : MpComGetLink;
END_VAR
(*------------------------------------------------------------------------------------------------------------------------------------------------------------------------------------------------------------------------*)
(*Error numbers*)
VAR CONSTANT
	ERR_REC_TOO_MANY_CLIENTS : DINT := 50010; (*More than 3 clients try to connect to recipe management*)
	ERR_REC_NAME_EMPTY : DINT := 50100; (*Recipe name is empty*)
	ERR_REC_NAME_EXISTS : DINT := 50101; (*Recipe name already exists*)
	ERR_REC_NAME_LOST : DINT := 50102; (*Recipe name was not found*)
	ERR_REC_NAME_LENGTH : DINT := 50103; (*One or more recipe names exceeds maximum length*)
END_VAR
VAR
	ERR_REC_DEV_NAME_EMPTY : DINT := 50110; (*Device name is empty*)
END_VAR
VAR CONSTANT
	ERR_REC_VAR_NAME_EMPTY : DINT := 50120; (*Variable name is empty*)
	ERR_REC_NOT_INITIALIZED : DINT := 50130; (*Recipemanagement is not initialized*)
	ERR_REC_REC_NUM : DINT := 50140; (*Maximum number of recipes reached*)
	ERR_REC_TASK_NAME : DINT := 50150; (*Task name is incorrect*)
END_VAR
VAR
	ERR_MEM_ALLOC : UINT := 50300; (*Memory allocation for file upload and download failed*)
	ERR_MEM_DOWNLOAD : UINT := 50310; (*Size of download file exceeds maximum*)
	ERR_TIMEOUT_DOWNLOAD : UINT := 50320; (*Download response timed out*)
	ERR_POS_NAME_UPLOAD : UINT := 50400; (*Can not find filename in upload response*)
	ERR_SIZE_NAME_UPLOAD : UINT := 50401; (*Can not determine end of filename in upload response*)
	ERR_LEN_NAME_UPLOAD : UINT := 50402; (*Filename is too long in upload response*)
	ERR_POS_DATA_UPLOAD : UINT := 50403; (*Can not find data in upload response*)
	ERR_SIZE_DATA_UPLOAD : UINT := 50404; (*Can not determine end of data in upload response*)
	ERR_MEM_UPLOAD : UINT := 50410; (*Size of upload file exceeds maximum size*)
	ERR_UNICODE_UPLOAD : UINT := 50420; (*Upload is not supported when unicode is used*)
END_VAR
```

#### LocalFunctions.fun - Local function definition
```iecst
FUNCTION CreateError : recSTATE
	VAR_INPUT
		RECIPE : REFERENCE TO recMAIN;
		No : DINT;
		Text : WSTRING[200];
		State : recSTATE;
	END_VAR
END_FUNCTION

FUNCTION CreateMessage : BOOL
	VAR_INPUT
		TargetString : UDINT;
		Text : UDINT;
		RecipeName : UDINT;
		VisuSlotID : USINT;
	END_VAR
	VAR
		VisuSlotIDStr : WSTRING[5];
		tmpWStr1 : WSTRING[200];
	END_VAR
END_FUNCTION

FUNCTION FindRecName : UINT
	VAR_INPUT
		RECIPE : REFERENCE TO recMAIN;
		RecipeName : WSTRING[REC_NAME_LENGTH];
	END_VAR
	VAR
		idx : UINT;
	END_VAR
END_FUNCTION

FUNCTION InsertRecName : UINT
	VAR_INPUT
		RECIPE : REFERENCE TO recMAIN;
		new_name : WSTRING[REC_NAME_LENGTH];
		new_id : STRING[REC_NAME_LENGTH];
	END_VAR
	VAR
		idx : INT;
		idy : INT;
		lSort : DINT;
		lValue : DINT;
		tmpSTR : STRING[REC_NAME_LENGTH];
	END_VAR
END_FUNCTION

FUNCTION RemoveRecName : BOOL
	VAR_INPUT
		RECIPE : REFERENCE TO recMAIN;
		RecipeIndex : UINT;
	END_VAR
END_FUNCTION

FUNCTION IsInstrW : BOOL
	VAR_INPUT
		string1 : UDINT;
		string2 : UDINT;
	END_VAR
	VAR
		idx : UDINT;
	END_VAR
END_FUNCTION

FUNCTION WorkingStatus : USINT
	VAR_INPUT
		RECIPE : REFERENCE TO recMAIN;
		str : UDINT;
		animation : USINT;
	END_VAR
END_FUNCTION

FUNCTION WString2DataProvider : BOOL
	VAR_INPUT
		SourceString : UDINT;
		TargetString : UDINT;
	END_VAR
END_FUNCTION

FUNCTION ReplaceString : BOOL
	VAR_INPUT
		dataSTR : UDINT;
		searchSTR : UDINT;
		replaceSTR : UDINT;
		first : BOOL;
	END_VAR
	VAR
		idx : UDINT;
	END_VAR
END_FUNCTION

FUNCTION FindInMem : DINT
	VAR_INPUT
		data1 : UDINT;
		len1 : UDINT;
		data2 : UDINT;
		len2 : UDINT;
		direction : BOOL;
	END_VAR
	VAR
		idx : UDINT;
	END_VAR
END_FUNCTION
```

#### LocalFunctions.st - Local function code
```iecst
//******************************************************************************************************
// Find recipe name
//******************************************************************************************************
FUNCTION FindRecName
	// Check if recipe name exists
	IF(RECIPE.DAT.RecipeNum > 0) THEN
		FOR idx:=0 TO RECIPE.DAT.RecipeNum - 1 DO
			IF(RECIPE.DAT.RecipeNames[idx] = RecipeName) THEN
				FindRecName := idx;
				RETURN;
			END_IF
		END_FOR;
	END_IF
	FindRecName := REC_DOES_NOT_EXIST;
END_FUNCTION

//******************************************************************************************************
// Create mappView data provider string
//******************************************************************************************************
FUNCTION WString2DataProvider
	brwcscpy(TargetString, ADR("{$"value$":$""));
	brwcscat(TargetString, SourceString);
	brwcscat(TargetString, ADR("$",$"text$":$""));
	brwcscat(TargetString, SourceString);
	brwcscat(TargetString, ADR("$"}"));

	WString2DataProvider := TRUE;
END_FUNCTION

//******************************************************************************************************
// Create error
//******************************************************************************************************
FUNCTION CreateError
	RECIPE.ERR.No := No;
	RECIPE.ERR.State := State;
	RECIPE.ERR.Text := Text;
	CreateError := REC_ERROR;
END_FUNCTION

//******************************************************************************************************
// Create status meesage
//******************************************************************************************************
FUNCTION CreateMessage
	brwcscpy(ADR(tmpWStr1), Text);
	brwcscat(ADR(tmpWStr1), ADR(" "));
	brwcscat(ADR(tmpWStr1), RecipeName);
	brwcscat(ADR(tmpWStr1), ADR(" on web client ID "));
	VisuSlotIDStr := DINT_TO_WSTRING(VisuSlotID);
	brwcscat(ADR(tmpWStr1), ADR(VisuSlotIDStr));
	brwcscpy(TargetString, ADR(tmpWStr1));

	CreateMessage := TRUE;
END_FUNCTION

//******************************************************************************************************
// Working status
//******************************************************************************************************
FUNCTION WorkingStatus
	animation := animation+1;

	IF (animation = 80) THEN
		animation := 0;
	END_IF

	brsmemset(ADR(RECIPE.DAT.Status), 0, SIZEOF(RECIPE.DAT.Status));
	brwcscpy(ADR(RECIPE.DAT.Status), str);
	CASE(animation) OF
		0..19	: brwcscat(ADR(RECIPE.DAT.Status), ADR("/"));
		20..39	: brwcscat(ADR(RECIPE.DAT.Status), ADR("-"));
		40..59	: brwcscat(ADR(RECIPE.DAT.Status), ADR("\"));
		60..79	: brwcscat(ADR(RECIPE.DAT.Status), ADR("|"));
	END_CASE;
	WorkingStatus := animation;
END_FUNCTION

//******************************************************************************************************
// Remove recipe name from list
//******************************************************************************************************
FUNCTION RemoveRecName
	// Remove name from recipe list
	IF(RecipeIndex < REC_REC_NUM) THEN
		brsmemmove(ADR(RECIPE.DAT.RecipeNames[RecipeIndex]),ADR(RECIPE.DAT.RecipeNames[RecipeIndex+1]), (REC_REC_NUM - RecipeIndex) * SIZEOF(RECIPE.DAT.RecipeNames[0]));
		brsmemmove(ADR(RECIPE.DAT.RecipeIDs[RecipeIndex]),ADR(RECIPE.DAT.RecipeIDs[RecipeIndex+1]), (REC_REC_NUM - RecipeIndex) * SIZEOF(RECIPE.DAT.RecipeIDs[0]));
	END_IF
	brsmemset(ADR(RECIPE.DAT.RecipeNames[REC_REC_NUM]), 0, SIZEOF(ADR(RECIPE.DAT.RecipeNames[0])));
	brsmemset(ADR(RECIPE.DAT.RecipeIDs[REC_REC_NUM]), 0, SIZEOF(ADR(RECIPE.DAT.RecipeIDs[0])));
	RECIPE.DAT.RecipeNum := RECIPE.DAT.RecipeNum - 1;
	RemoveRecName := TRUE;
END_FUNCTION

//******************************************************************************************************
// Insert new recipe name
//******************************************************************************************************
FUNCTION InsertRecName
	// Sort recipes names numeric
	IF(REC_SORT_NUMERIC) THEN
		IF(RECIPE.DAT.RecipeNum > 0) THEN
			brwcsconv(ADR(tmpSTR), ADR(new_name), brwUCtoU8);
			lValue := brsatoi(ADR(tmpSTR));
			FOR idx:=0 TO UINT_TO_INT(RECIPE.DAT.RecipeNum - 1) DO
				brwcsconv(ADR(tmpSTR), ADR(RECIPE.DAT.RecipeNames[idx]), brwUCtoU8);
				lSort := brsatoi(ADR(tmpSTR));
				IF(lValue < lSort) THEN
					EXIT;
				END_IF
			END_FOR;
		END_IF
	// Sort recipes names alphabetic
	ELSE
		// Set up start values for iteration
		IF (RECIPE.DAT.RecipeNum <> 0) THEN
			idy := RECIPE.DAT.RecipeNum - 1;
		END_IF
		idx := idy;

		// Start iteration	search
		WHILE (idy > 1) DO
			// Check current entry
			lSort := brwcscmp(ADR(new_name), ADR(RECIPE.DAT.RecipeNames[idy]));
			// Solve new search range
			IF (idy MOD 2 = 0) THEN
				idy := idy / 2;
			ELSE
				idy := idy / 2 + 1;
			END_IF
			// New range is lower or higher than current
			IF (lSort > 0) THEN
				idx := idx + idy;
				IF (idx > UINT_TO_INT(RECIPE.DAT.RecipeNum)) THEN
					idx := RECIPE.DAT.RecipeNum;
				END_IF
			ELSE
				idx := idx - idy;
				IF (idx < 1) THEN
					idx := 1;
				END_IF
			END_IF
		END_WHILE;

		// New entry is this, next or previous
		lSort := brwcscmp(ADR(new_name), ADR(RECIPE.DAT.RecipeNames[idx]));
		IF (lSort > 0 AND idx <> UINT_TO_INT(RECIPE.DAT.RecipeNum)) THEN
			idx := idx +1;
		ELSIF (idx > 0) THEN
			lSort := brwcscmp(ADR(new_name), ADR(RECIPE.DAT.RecipeNames[idx-1]));
			IF (lSort < 0) THEN
				idx := idx - 1;
			END_IF
		END_IF
	END_IF

	// Move all data entrys backwards and fill in new entry
	IF(idx < REC_REC_NUM) THEN
		brsmemmove(ADR(RECIPE.DAT.RecipeNames[idx+1]),ADR(RECIPE.DAT.RecipeNames[idx]), (RECIPE.DAT.RecipeNum - idx) * SIZEOF(RECIPE.DAT.RecipeNames[1]));
		brsmemmove(ADR(RECIPE.DAT.RecipeIDs[idx+1]),ADR(RECIPE.DAT.RecipeIDs[idx]), (RECIPE.DAT.RecipeNum - idx) * SIZEOF(RECIPE.DAT.RecipeIDs[1]));
	END_IF
	brwcscpy(ADR(RECIPE.DAT.RecipeNames[idx]), ADR(new_name));
	brsstrcpy(ADR(RECIPE.DAT.RecipeIDs[idx]), ADR(new_id));

	RECIPE.DAT.RecipeNum := RECIPE.DAT.RecipeNum + 1;
	InsertRecName := idx;
END_FUNCTION

//******************************************************************************************************
// Is second string in first string
//******************************************************************************************************
FUNCTION IsInstrW
	IF (brwcslen(string1) >= brwcslen(string2)) THEN
		FOR idx:=0 TO brwcslen(string1) - brwcslen(string2) DO
			IF (brwcsncmp(string1 + (2*idx), string2, brwcslen(string2)) = 0) THEN
				IsInstrW := TRUE;
				EXIT;
			END_IF
		END_FOR;
	END_IF
END_FUNCTION

//******************************************************************************************************
// Find second data in first data
//******************************************************************************************************
FUNCTION FindInMem
	IF (len1 > len2) THEN
		FOR idx:=0 TO len1 - len2 DO
			IF (brsmemcmp(data1 + idx, data2, len2) = 0) THEN
				FindInMem := idx;
				EXIT;
			END_IF
		END_FOR;
	END_IF
END_FUNCTION

//******************************************************************************************************
// Find and replace string
//******************************************************************************************************
FUNCTION ReplaceString
	IF (brsstrlen(dataSTR) >= brsstrlen(searchSTR)) THEN
		FOR idx:=0 TO brsstrlen(dataSTR) - brsstrlen(searchSTR) DO
			IF (brsmemcmp(dataSTR + idx, searchSTR, brsstrlen(searchSTR)) = 0) THEN
				// Move data around
				brsmemmove(dataSTR + idx + brsstrlen(replaceSTR), dataSTR + idx + brsstrlen(searchSTR), brsstrlen(dataSTR) - brsstrlen(searchSTR) + 1);
				brsmemcpy(dataSTR + idx, replaceSTR, brsstrlen(replaceSTR));
				// Set found flag and exit if only one hit is needed
				ReplaceString := TRUE;
				IF(first) THEN
					EXIT;
				END_IF
				// Correct index for next search
				IF(brsstrlen(replaceSTR) > 0) THEN
					idx := idx + brsstrlen(replaceSTR);
				END_IF
				idx := idx - 1;
				// Exit if no data is left
				IF (brsstrlen(dataSTR) = 0 OR brsstrlen(dataSTR) < brsstrlen(searchSTR)) THEN
					EXIT;
				END_IF
			END_IF
		END_FOR;
	END_IF
END_FUNCTION
```

### Program Logical/mappRecipe/YourTask (IEC)

#### Main.st - Init, cyclic, exit code
```iecst
// --------------------------------------------------------------------------------------------------------------------
// Use this task to add your own code for recipe managment
// --------------------------------------------------------------------------------------------------------------------
PROGRAM _INIT
	// Sample recipe data, the global array REC_VAR_LIST define what variables belong to a recipe
	MaschineData;
	ProductID := 'Cookies';
	CustomerID := 'B&R';

END_PROGRAM

PROGRAM _CYCLIC
	(* Insert code here *)

END_PROGRAM

PROGRAM _EXIT
	(* Insert code here *)

END_PROGRAM
```

#### YourTypes.typ - Local data types
```iecst
(*Structure that contains the recipe variables*)

TYPE
	recVariable : 	STRUCT
		Temperature1 : INT := 11;
		Temperature2 : INT := 22;
		MotorSpeed : DINT := 33;
		Position : REAL := 44.55;
	END_STRUCT;
END_TYPE
```

#### YourVariables.var - Local variables
```iecst
VAR
	MaschineData : recVariable; (*Structure that contains the recipe variables*)
	ProductID : STRING[80];
	CustomerID : STRING[80];
	cmd_create : BOOL;
	tmpStr1 : STRING[80];
	tmpStr2 : STRING[80];
	counter : UDINT;
	idx : UINT;
END_VAR
```

### changelog.txt
```
Version 0.8
- Changed some parameters to constants
- Simplified configuration
- Added better error messages
- Added the possibility to define multiple variables

Version 0.7
- Fixed recipe view does not show correct data on double click or command view
- Fixed ReplaceString function call

Version 0.6
- Code cleanup
- Option to sort recipe names as numeric values instead of alphabetic
- Renamed web controls to avoid conflicts with other samples
- Fixed download not working when downloading the same file again
- Fixed upload not working with large files > 1 MB

Version 0.5
- Added support for recipe upload over mappView
- Fixed renaming recipes in ASCII mode

Version 0.4
- Added support for recipe download over mappView
- Removed view file status message
- Code cleanup

Version 0.3
- Added categories to mapp function blocks to seperate recipe data
- Added function to view files by double click or command
- Removed obsolete constants

Version 0.2
- Added message box before saving or deleting a recipe
- Fixed filter compare too short
- Added exit function
- Code cleanup

Version 0.1
- First public release
```

### Types.typ - not listed in the package file held
```iecst
(*------------------------------------------------------------------------------------------------------------------------------------------------------------------------------------------------------------------------*)
(*Global enumerations*)

TYPE
	recSTATE :
		( (*Recipe management state machine*)
		REC_WAIT,
		REC_REG_NAME,
		REC_REG_VAR,
		REC_CREATE_DIR,
		REC_READ_DIR,
		REC_READ_DIR_1,
		REC_READ_DIR_2,
		REC_READ_DIR_3,
		REC_GEN_FILE_NAME,
		REC_LOAD_SAVE,
		REC_DELETE,
		REC_RENAME,
		REC_VIEW,
		REC_DOWNLOAD,
		REC_DOWNLOAD_1,
		REC_DOWNLOAD_2,
		REC_DOWNLOAD_3,
		REC_DOWNLOAD_4,
		REC_UPLOAD,
		REC_UPLOAD_1,
		REC_UPLOAD_2,
		REC_UPLOAD_3,
		REC_UPLOAD_4,
		REC_UPLOAD_5,
		REC_UPLOAD_6,
		REC_ERROR
		);
	recTYPE :
		(
		typeCSV,
		typeXML
		);
END_TYPE

(*------------------------------------------------------------------------------------------------------------------------------------------------------------------------------------------------------------------------*)
(*Global structure*)

TYPE
	recERR : 	STRUCT  (*Recipe management error structure*)
		Text : WSTRING[200]; (* Error text *)
		No : DINT; (* Error number *)
		State : recSTATE; (* Error step *)
	END_STRUCT;
	recCMD : 	STRUCT  (*Recipe management command structure*)
		Init : BOOL := TRUE; (*Init recipes managment*)
		New : BOOL; (*Create new recipe*)
		Load : BOOL; (*Load recipe*)
		Save : BOOL; (*Save recipe*)
		View : BOOL; (*View recipe*)
		Rename : BOOL; (*Rename recipe*)
		Delete : BOOL; (*Delete recipe*)
		Download : BOOL; (*Download recipe*)
		Upload : BOOL; (*Upload recipe*)
		ErrorReset : BOOL; (*Reset pending errors*)
	END_STRUCT;
	recPAR : 	STRUCT  (*Recipe management parameter structure*)
		RecipeVariable : STRING[200]; (*Name of the variable where the data is stored*)
		RecipeName : WSTRING[REC_NAME_LENGTH]; (*Recipe name*)
		RecipeNameNew : WSTRING[REC_NAME_LENGTH]; (*New recipe name*)
		RecipeID : STRING[REC_NAME_LENGTH]; (*File name of the recipe*)
		RecipeDirectory : STRING[200]; (*Recipe directory*)
		DeviceName : STRING[100]; (*Device name where the recipes are stored*)
		MpLink : MpComIdentType; (*MpLink from mappRecipe*)
		Initialized : BOOL; (*Indicates that recipe management was initialized*)
		VisuSlotID : USINT; (*ID for connected web connection*)
		VisuEnableCommand : BOOL;
	END_STRUCT;
	recDAT : 	STRUCT  (*Recipe management data structure*)
		RecipeNames : ARRAY[0..REC_MAX_NUM]OF WSTRING[REC_NAME_LENGTH]; (*Recipe unicode names*)
		RecipeIDs : ARRAY[0..REC_MAX_NUM]OF STRING[REC_NAME_LENGTH]; (*File name of the recipes*)
		RecipeNum : UINT; (*Number of recipes*)
		Status : WSTRING[100]; (*Shows the result of the last command*)
	END_STRUCT;
	recVIS : 	STRUCT  (*Recipe management visualization structure*)
		RecipeNames : ARRAY[0..REC_MAX_NUM]OF WSTRING[REC_VIS_LENGTH]; (*Recipe names as mappView data provider*)
		RecipeNum : UINT; (*Number of visible recipes*)
		RecipeFilter : WSTRING[REC_NAME_LENGTH]; (*Only show recipes that fit this pattern*)
		RecipeSelect : WSTRING[REC_NAME_LENGTH]; (*Select recipe in listbox after command new or rename*)
		DownloadFileUrl : STRING[REC_NAME_LENGTH]; (*URL used with recipe download*)
		UploadOverwriteRequest : BOOL; (*Show message box to overwrite file*)
		UploadOverwriteResponse : USINT; (*Response from message box overwrite file*)
		ReloadUpload : BOOL; (*Reload upload button*)
		RecipeDoubleClick : USINT; (*Track double click event*)
		ViewFilePath : STRING[REC_VIS_LENGTH]; (*Full path for viewing file*)
		ViewFile : BOOL; (*Trigger that opens the fly out window when viewing recipes*)
		ShowMessageBoxError : BOOL; (*Show message box on error*)
	END_STRUCT;
	recMAIN : 	STRUCT  (*Recipe management main structure*)
		CMD : recCMD; (* Command structure *)
		PAR : recPAR; (* Parameter structure *)
		DAT : recDAT; (*Data structure*)
		VIS : ARRAY[0..REC_MAX_CLIENTS_ID]OF recVIS; (*Visualization structure*)
		ERR : recERR; (* Error structure *)
	END_STRUCT;
END_TYPE

(*------------------------------------------------------------------------------------------------------------------------------------------------------------------------------------------------------------------------*)
(*Structure that contains the recipe variables*)

TYPE
	recVariable : 	STRUCT
		Temperature1 : INT := 11;
		Temperature2 : INT := 22;
		MotorSpeed : DINT := 33;
		Position : REAL := 44.55;
	END_STRUCT;
END_TYPE
```
